C09150=1163.672,78.044,-51.262,-179.316,6.272,148.934
C09151=1163.677,77.794,-51.245,-179.319,6.271,148.934
C09152=1163.682,77.544,-51.228,-179.321,6.270,148.935
C09153=1163.686,77.295,-51.210,-179.324,6.269,148.935
C09154=1163.692,77.046,-51.193,-179.327,6.267,148.936
C09155=1163.696,76.797,-51.177,-179.329,6.266,148.936
C09156=1163.702,76.547,-51.159,-179.332,6.265,148.937
C09157=1163.707,76.298,-51.141,-179.335,6.263,148.937
C09158=1163.711,76.048,-51.125,-179.338,6.263,148.938
C09159=1163.717,75.799,-51.108,-179.340,6.261,148.938
C09160=1163.721,75.550,-51.091,-179.342,6.260,148.939
C09161=1163.727,75.300,-51.074,-179.346,6.259,148.939
C09162=1163.731,75.050,-51.057,-179.348,6.258,148.940
C09163=1163.736,74.801,-51.039,-179.351,6.257,148.940
C09164=1163.741,74.553,-51.023,-179.353,6.256,148.941
C09165=1163.746,74.303,-51.006,-179.356,6.254,148.941
C09166=1163.751,74.053,-50.989,-179.359,6.254,148.942
C09167=1163.755,73.804,-50.972,-179.361,6.252,148.942
C09168=1163.761,73.555,-50.955,-179.364,6.252,148.943
C09169=1163.766,73.305,-50.939,-179.367,6.250,148.944
C09170=1163.771,73.055,-50.922,-179.369,6.249,148.944
C09171=1163.775,72.807,-50.904,-179.372,6.248,148.945
C09172=1163.781,72.557,-50.887,-179.374,6.247,148.945
C09173=1163.785,72.308,-50.871,-179.377,6.246,148.946
C09174=1163.790,72.058,-50.854,-179.380,6.244,148.946
C09175=1163.796,71.809,-50.837,-179.383,6.243,148.947
C09176=1163.800,71.560,-50.820,-179.385,6.242,148.947
C09177=1163.805,71.310,-50.803,-179.388,6.241,148.948
C09178=1163.810,71.061,-50.786,-179.391,6.239,148.948
C09179=1163.815,70.812,-50.770,-179.393,6.239,148.949
C09180=1163.820,70.562,-50.753,-179.396,6.237,148.949
C09181=1163.824,70.313,-50.736,-179.398,6.236,148.950
C09182=1163.830,70.064,-50.720,-179.401,6.235,148.950
C09183=1163.835,69.814,-50.703,-179.404,6.234,148.951
C09184=1163.839,69.564,-50.686,-179.406,6.233,148.951
C09185=1163.844,69.316,-50.670,-179.409,6.232,148.952
C09186=1163.850,69.065,-50.653,-179.412,6.230,148.952
C09187=1163.854,68.816,-50.636,-179.414,6.230,148.953
C09188=1163.859,68.567,-50.620,-179.417,6.228,148.954
C09189=1163.865,68.317,-50.603,-179.419,6.227,148.954
C09190=1163.869,68.068,-50.586,-179.423,6.226,148.955
C09191=1163.874,67.819,-50.570,-179.425,6.225,148.955
C09192=1163.879,67.569,-50.553,-179.427,6.225,148.956
C09193=1163.884,67.320,-50.536,-179.430,6.223,148.956
C09194=1163.889,67.071,-50.520,-179.433,6.222,148.957
C09195=1163.894,66.821,-50.504,-179.435,6.221,148.957
C09196=1163.900,66.572,-50.487,-179.438,6.220,148.958
C09197=1163.904,66.322,-50.470,-179.441,6.219,148.958
C09198=1163.909,66.073,-50.453,-179.443,6.218,148.959
C09199=1163.914,65.824,-50.437,-179.446,6.216,148.959
C09200=1163.919,65.574,-50.420,-179.448,6.215,148.960
C09201=1163.924,65.325,-50.404,-179.452,6.214,148.961
C09202=1163.929,65.075,-50.388,-179.454,6.213,148.961
C09203=1163.933,64.826,-50.371,-179.457,6.212,148.962
C09204=1163.938,64.577,-50.355,-179.459,6.211,148.962
C09205=1163.944,64.327,-50.338,-179.462,6.209,148.962
C09206=1163.949,64.078,-50.322,-179.464,6.209,148.963
C09207=1163.953,63.828,-50.305,-179.467,6.207,148.964
C09208=1163.958,63.579,-50.288,-179.470,6.207,148.964
C09209=1163.963,63.329,-50.273,-179.472,6.206,148.965
C09210=1163.968,63.080,-50.256,-179.475,6.205,148.965
C09211=1163.974,62.831,-50.239,-179.477,6.204,148.966
C09212=1163.978,62.581,-50.223,-179.481,6.202,148.966
C09213=1163.983,62.332,-50.207,-179.483,6.202,148.967
C09214=1163.988,62.082,-50.190,-179.485,6.200,148.967
C09215=1163.993,61.833,-50.175,-179.488,6.199,148.968
C09216=1163.998,61.584,-50.158,-179.491,6.198,148.968
C09217=1164.004,61.334,-50.141,-179.493,6.197,148.969
C09218=1164.008,61.084,-50.125,-179.496,6.195,148.969
C09219=1164.013,60.836,-50.109,-179.499,6.195,148.970
C09220=1164.018,60.585,-50.093,-179.501,6.194,148.971
C09221=1164.023,60.337,-50.077,-179.504,6.193,148.971
C09222=1164.028,60.087,-50.060,-179.506,6.192,148.972
C09223=1164.033,59.837,-50.044,-179.510,6.191,148.972
C09224=1164.038,59.588,-50.028,-179.512,6.190,148.973
C09225=1164.043,59.339,-50.012,-179.514,6.188,148.973
C09226=1164.047,59.089,-49.996,-179.517,6.188,148.974
C09227=1164.053,58.840,-49.980,-179.519,6.187,148.974
C09228=1164.057,58.591,-49.963,-179.522,6.185,148.975
C09229=1164.063,58.341,-49.948,-179.525,6.185,148.975
C09230=1164.068,58.091,-49.930,-179.528,6.183,148.976
C09231=1164.073,57.843,-49.914,-179.530,6.182,148.977
C09232=1164.078,57.592,-49.898,-179.533,6.181,148.977
C09233=1164.083,57.343,-49.883,-179.535,6.180,148.978
C09234=1164.088,57.094,-49.866,-179.538,6.180,148.978
C09235=1164.093,56.844,-49.850,-179.541,6.178,148.979
C09236=1164.098,56.595,-49.834,-179.543,6.178,148.979
C09237=1164.103,56.345,-49.818,-179.546,6.176,148.980
C09238=1164.108,56.097,-49.802,-179.549,6.175,148.981
C09239=1164.113,55.846,-49.786,-179.551,6.174,148.981
C09240=1164.118,55.598,-49.770,-179.554,6.173,148.981
C09241=1164.123,55.348,-49.754,-179.556,6.172,148.982
C09242=1164.128,55.098,-49.738,-179.559,6.171,148.982
C09243=1164.132,54.849,-49.722,-179.562,6.170,148.983
C09244=1164.137,54.600,-49.706,-179.564,6.169,148.984
C09245=1164.143,54.331,-49.689,-179.567,6.168,148.984
C09246=1164.148,54.063,-49.672,-179.570,6.167,148.985
C09247=1164.153,53.793,-49.655,-179.572,6.166,148.985
C09248=1164.159,53.526,-49.637,-179.576,6.165,148.986
C09249=1164.164,53.276,-49.622,-179.578,6.164,148.987
C09250=1164.169,53.026,-49.606,-179.581,6.162,148.987
C09251=1164.174,52.777,-49.589,-179.584,6.162,148.988
C09252=1164.179,52.528,-49.574,-179.586,6.161,148.988
C09253=1164.184,52.278,-49.558,-179.589,6.159,148.989
C09254=1164.189,52.028,-49.542,-179.591,6.159,148.989
C09255=1164.194,51.779,-49.526,-179.593,6.158,148.990
C09256=1164.198,51.530,-49.511,-179.597,6.157,148.990
C09257=1164.204,51.280,-49.495,-179.599,6.156,148.991
C09258=1164.209,51.030,-49.479,-179.602,6.155,148.992
C09259=1164.214,50.782,-49.463,-179.604,6.154,148.992
C09260=1164.219,50.532,-49.447,-179.607,6.153,148.993
C09261=1164.224,50.282,-49.431,-179.610,6.151,148.993
C09262=1164.229,50.033,-49.416,-179.612,6.151,148.994
C09263=1164.234,49.784,-49.400,-179.614,6.150,148.994
C09264=1164.238,49.534,-49.384,-179.618,6.149,148.995
C09265=1164.244,49.285,-49.368,-179.620,6.148,148.995
C09266=1164.249,49.035,-49.353,-179.623,6.147,148.996
C09267=1164.253,48.785,-49.337,-179.625,6.146,148.996
C09268=1164.259,48.536,-49.322,-179.628,6.145,148.997
C09269=1164.264,48.287,-49.305,-179.630,6.144,148.998
C09270=1164.268,48.037,-49.290,-179.633,6.143,148.998
C09271=1164.274,47.788,-49.274,-179.635,6.142,148.999
C09272=1164.279,47.539,-49.259,-179.639,6.141,148.999
C09273=1164.284,47.289,-49.243,-179.641,6.140,149.000
C09274=1164.289,47.039,-49.227,-179.643,6.140,149.000
C09275=1164.294,46.790,-49.212,-179.646,6.138,149.001
C09276=1164.299,46.541,-49.197,-179.649,6.137,149.002
C09277=1164.304,46.291,-49.181,-179.651,6.137,149.002
C09278=1164.309,46.041,-49.165,-179.654,6.135,149.003
C09279=1164.314,45.792,-49.150,-179.656,6.134,149.003
C09280=1164.319,45.543,-49.135,-179.659,6.134,149.004
C09281=1164.323,45.293,-49.118,-179.662,6.132,149.004
C09282=1164.329,45.044,-49.102,-179.664,6.132,149.005
C09283=1164.333,44.795,-49.087,-179.666,6.131,149.005
C09284=1164.339,44.545,-49.072,-179.670,6.130,149.006
C09285=1164.344,44.295,-49.056,-179.672,6.129,149.006
C09286=1164.348,44.046,-49.041,-179.674,6.128,149.007
C09287=1164.354,43.796,-49.026,-179.677,6.127,149.008
C09288=1164.359,43.547,-49.010,-179.680,6.126,149.008
C09289=1164.364,43.298,-48.995,-179.682,6.125,149.009
C09290=1164.369,43.047,-48.980,-179.685,6.124,149.009
C09291=1164.374,42.798,-48.964,-179.687,6.123,149.010
C09292=1164.379,42.549,-48.949,-179.690,6.123,149.011
C09293=1164.384,42.300,-48.933,-179.693,6.121,149.011
C09294=1164.389,42.050,-48.918,-179.695,6.121,149.012
C09295=1164.394,41.800,-48.902,-179.698,6.120,149.012
C09296=1164.399,41.551,-48.887,-179.701,6.118,149.013
C09297=1164.404,41.302,-48.872,-179.703,6.118,149.013
C09298=1164.409,41.052,-48.856,-179.706,6.117,149.014
C09299=1164.414,40.803,-48.842,-179.708,6.115,149.014
C09300=1164.419,40.553,-48.826,-179.711,6.115,149.015
C09301=1164.424,40.303,-48.810,-179.713,6.114,149.015
C09302=1164.429,40.054,-48.795,-179.716,6.113,149.016
C09303=1164.434,39.805,-48.780,-179.719,6.112,149.017
C09304=1164.439,39.556,-48.765,-179.721,6.111,149.017
C09305=1164.445,39.306,-48.750,-179.724,6.111,149.018
C09306=1164.449,39.057,-48.735,-179.727,6.109,149.018
C09307=1164.454,38.806,-48.719,-179.729,6.109,149.019
C09308=1164.459,38.557,-48.704,-179.731,6.108,149.019
C09309=1164.464,38.308,-48.688,-179.735,6.107,149.020
C09310=1164.470,38.058,-48.674,-179.737,6.106,149.021
C09311=1164.474,37.809,-48.659,-179.739,6.105,149.021
C09312=1164.480,37.559,-48.643,-179.742,6.104,149.022
C09313=1164.484,37.310,-48.628,-179.745,6.103,149.022
C09314=1164.490,37.060,-48.613,-179.747,6.102,149.023
C09315=1164.494,36.811,-48.598,-179.750,6.102,149.023
C09316=1164.500,36.561,-48.582,-179.752,6.100,149.024
C09317=1164.505,36.311,-48.568,-179.755,6.100,149.025
C09318=1164.509,36.062,-48.553,-179.757,6.099,149.025
C09319=1164.515,35.813,-48.537,-179.760,6.098,149.026
C09320=1164.519,35.564,-48.522,-179.763,6.097,149.026
C09321=1164.525,35.314,-48.507,-179.765,6.096,149.027
C09322=1164.530,35.065,-48.492,-179.767,6.095,149.027
C09323=1164.535,34.815,-48.478,-179.771,6.094,149.028
C09324=1164.540,34.566,-48.463,-179.773,6.094,149.029
C09325=1164.545,34.316,-48.447,-179.775,6.093,149.029
C09326=1164.550,34.066,-48.433,-179.778,6.092,149.030
C09327=1164.555,33.817,-48.418,-179.781,6.091,149.030
C09328=1164.560,33.567,-48.402,-179.783,6.090,149.031
C09329=1164.565,33.318,-48.387,-179.786,6.089,149.031
C09330=1164.570,33.068,-48.372,-179.789,6.088,149.032
C09331=1164.575,32.818,-48.358,-179.791,6.087,149.032
C09332=1164.580,32.569,-48.343,-179.794,6.087,149.033
C09333=1164.585,32.319,-48.328,-179.796,6.086,149.034
C09334=1164.590,32.070,-48.313,-179.799,6.085,149.034
C09335=1164.595,31.821,-48.298,-179.801,6.084,149.035
C09336=1164.600,31.571,-48.283,-179.804,6.083,149.035
C09337=1164.605,31.322,-48.268,-179.806,6.082,149.036
C09338=1164.611,31.072,-48.253,-179.809,6.081,149.037
C09339=1164.615,30.823,-48.238,-179.812,6.081,149.037
C09340=1164.620,30.573,-48.224,-179.814,6.080,149.038
C09341=1164.625,30.324,-48.209,-179.817,6.079,149.038
C09342=1164.631,30.074,-48.194,-179.819,6.078,149.039
C09343=1164.635,29.825,-48.179,-179.822,6.077,149.039
C09344=1164.640,29.575,-48.165,-179.824,6.076,149.040
C09345=1164.646,29.325,-48.150,-179.827,6.076,149.041
C09346=1164.651,29.076,-48.135,-179.830,6.074,149.041
C09347=1164.655,28.827,-48.120,-179.832,6.074,149.042
C09348=1164.661,28.577,-48.105,-179.834,6.073,149.042
C09349=1164.666,28.308,-48.089,-179.837,6.072,149.043
C09350=1164.671,28.040,-48.073,-179.840,6.071,149.044
C09351=1164.677,27.770,-48.057,-179.843,6.071,149.044
C09352=1164.683,27.502,-48.042,-179.846,6.069,149.045
C09353=1164.688,27.253,-48.028,-179.848,6.068,149.045
C09354=1164.693,27.003,-48.013,-179.851,6.068,149.046
C09355=1164.698,26.754,-47.998,-179.853,6.067,149.046
C09356=1164.703,26.504,-47.983,-179.856,6.066,149.047
C09357=1164.708,26.254,-47.969,-179.859,6.065,149.048
C09358=1164.713,26.005,-47.954,-179.861,6.065,149.048
C09359=1164.718,25.755,-47.939,-179.863,6.064,149.049
C09360=1164.723,25.505,-47.925,-179.866,6.063,149.049
C09361=1164.728,25.256,-47.910,-179.869,6.062,149.050
C09362=1164.733,25.006,-47.896,-179.871,6.061,149.051
C09363=1164.738,24.757,-47.881,-179.874,6.060,149.051
C09364=1164.743,24.507,-47.867,-179.876,6.060,149.052
C09365=1164.749,24.258,-47.852,-179.879,6.059,149.052
C09366=1164.754,24.009,-47.838,-179.882,6.058,149.053
C09367=1164.759,23.759,-47.823,-179.884,6.057,149.054
C09368=1164.763,23.510,-47.808,-179.887,6.056,149.054
C09369=1164.768,23.260,-47.794,-179.889,6.056,149.055
C09370=1164.773,23.010,-47.780,-179.891,6.055,149.055
C09371=1164.779,22.760,-47.765,-179.895,6.054,149.056
C09372=1164.784,22.511,-47.751,-179.897,6.053,149.056
C09373=1164.788,22.262,-47.736,-179.899,6.052,149.057
C09374=1164.794,22.013,-47.722,-179.902,6.052,149.057
C09375=1164.799,21.763,-47.708,-179.904,6.051,149.058
C09376=1164.804,21.513,-47.693,-179.907,6.050,149.059
C09377=1164.809,21.263,-47.679,-179.910,6.049,149.059
C09378=1164.814,21.014,-47.665,-179.912,6.049,149.060
C09379=1164.818,20.765,-47.650,-179.914,6.048,149.060
C09380=1164.824,20.516,-47.636,-179.917,6.047,149.061
C09381=1164.830,20.266,-47.621,-179.920,6.046,149.061
C09382=1164.835,20.016,-47.607,-179.922,6.045,149.062
C09383=1164.840,19.766,-47.592,-179.925,6.045,149.063
C09384=1164.845,19.516,-47.578,-179.927,6.044,149.063
C09385=1164.850,19.267,-47.564,-179.930,6.043,149.064
C09386=1164.855,19.018,-47.550,-179.933,6.042,149.064
C09387=1164.860,18.768,-47.536,-179.935,6.041,149.065
C09388=1164.865,18.519,-47.521,-179.937,6.040,149.066
C09389=1164.870,18.269,-47.506,-179.940,6.040,149.066
C09390=1164.875,18.020,-47.492,-179.942,6.039,149.067
C09391=1164.880,17.771,-47.478,-179.945,6.039,149.067
C09392=1164.885,17.521,-47.464,-179.948,6.037,149.068
C09393=1164.890,17.271,-47.450,-179.950,6.037,149.068
C09394=1164.895,17.021,-47.435,-179.953,6.036,149.069
C09395=1164.900,16.772,-47.421,-179.955,6.035,149.070
C09396=1164.906,16.523,-47.407,-179.958,6.035,149.070
C09397=1164.911,16.273,-47.393,-179.960,6.034,149.071
C09398=1164.915,16.023,-47.379,-179.963,6.033,149.071
C09399=1164.920,15.774,-47.364,-179.965,6.032,149.072
C09400=1164.926,15.525,-47.350,-179.968,6.031,149.073
C09401=1164.931,15.275,-47.336,-179.971,6.031,149.073
C09402=1164.936,15.025,-47.322,-179.973,6.030,149.074
C09403=1164.941,14.775,-47.308,-179.976,6.030,149.074
C09404=1164.947,14.526,-47.294,-179.978,6.029,149.075
C09405=1164.951,14.276,-47.281,-179.981,6.027,149.076
C09406=1164.956,14.027,-47.266,-179.983,6.027,149.076
C09407=1164.961,13.777,-47.252,-179.986,6.026,149.077
C09408=1164.966,13.528,-47.238,-179.988,6.026,149.077
C09409=1164.971,13.278,-47.224,-179.991,6.025,149.078
C09410=1164.976,13.029,-47.210,-179.993,6.024,149.079
C09411=1164.982,12.780,-47.196,-179.995,6.024,149.079
C09412=1164.987,12.530,-47.181,-179.999,6.022,149.080
C09413=1164.992,12.279,-47.168,179.999,6.021,149.080
C09414=1164.996,12.030,-47.154,179.997,6.021,149.081
C09415=1165.002,11.781,-47.140,179.994,6.021,149.081
C09416=1165.007,11.531,-47.126,179.992,6.020,149.082
C09417=1165.012,11.282,-47.112,179.989,6.019,149.083
C09418=1165.017,11.033,-47.098,179.987,6.018,149.083
C09419=1165.023,10.782,-47.084,179.984,6.017,149.084
C09420=1165.028,10.533,-47.070,179.981,6.016,149.084
C09421=1165.032,10.284,-47.057,179.979,6.016,149.085
C09422=1165.037,10.034,-47.042,179.976,6.015,149.086
C09423=1165.043,9.784,-47.029,179.974,6.015,149.086
C09424=1165.048,9.535,-47.015,179.971,6.014,149.087
C09425=1165.053,9.285,-47.001,179.969,6.013,149.087
C09426=1165.057,9.036,-46.987,179.967,6.013,149.088
C09427=1165.063,8.786,-46.974,179.964,6.011,149.088
C09428=1165.068,8.536,-46.960,179.961,6.011,149.089
C09429=1165.073,8.287,-46.945,179.958,6.010,149.090
C09430=1165.079,8.038,-46.931,179.956,6.009,149.090
C09431=1165.083,7.788,-46.918,179.954,6.009,149.091
C09432=1165.089,7.539,-46.904,179.951,6.008,149.091
C09433=1165.094,7.289,-46.890,179.949,6.008,149.092
C09434=1165.099,7.039,-46.877,179.947,6.007,149.092
C09435=1165.104,6.790,-46.863,179.944,6.006,149.093
C09436=1165.109,6.540,-46.849,179.941,6.005,149.094
C09437=1165.114,6.290,-46.835,179.939,6.004,149.094
C09438=1165.120,6.041,-46.822,179.936,6.004,149.095
C09439=1165.124,5.791,-46.808,179.934,6.003,149.095
C09440=1165.130,5.542,-46.795,179.931,6.003,149.096
C09441=1165.135,5.292,-46.780,179.929,6.002,149.097
C09442=1165.139,5.042,-46.767,179.926,6.001,149.097
C09443=1165.145,4.793,-46.754,179.924,6.001,149.098
C09444=1165.150,4.543,-46.739,179.921,6.000,149.098
C09445=1165.155,4.294,-46.727,179.919,5.999,149.099
C09446=1165.160,4.044,-46.712,179.917,5.999,149.100
C09447=1165.166,3.795,-46.699,179.913,5.997,149.100
C09448=1165.170,3.545,-46.685,179.911,5.997,149.101
C09449=1165.175,3.295,-46.672,179.909,5.996,149.101
C09450=1165.181,3.046,-46.658,179.906,5.996,149.102
C09451=1165.185,2.797,-46.644,179.904,5.995,149.103
C09452=1165.191,2.547,-46.631,179.901,5.994,149.103
C09453=1165.196,2.278,-46.616,179.898,5.994,149.104
C09454=1165.201,2.008,-46.601,179.896,5.993,149.104
C09455=1165.207,1.739,-46.588,179.893,5.992,149.105
C09456=1165.213,1.470,-46.573,179.890,5.991,149.106
C09457=1165.217,1.220,-46.559,179.888,5.991,149.106
C09458=1165.223,0.971,-46.546,179.886,5.990,149.107
C09459=1165.228,0.720,-46.532,179.883,5.990,149.108
C09460=1165.233,0.471,-46.519,179.881,5.989,149.108
C09461=1165.238,0.221,-46.506,179.878,5.988,149.109
C09462=1165.243,-0.028,-46.492,179.876,5.988,149.109
C09463=1165.248,-0.278,-46.479,179.873,5.987,149.110
C09464=1165.254,-0.527,-46.465,179.871,5.987,149.111
C09465=1165.259,-0.777,-46.451,179.868,5.985,149.111
C09466=1165.264,-1.026,-46.439,179.865,5.985,149.112
C09467=1165.269,-1.276,-46.424,179.863,5.984,149.112
C09468=1165.274,-1.525,-46.412,179.860,5.983,149.113
C09469=1165.279,-1.775,-46.397,179.858,5.983,149.114
C09470=1165.284,-2.024,-46.385,179.856,5.982,149.114
C09471=1165.289,-2.275,-46.371,179.853,5.982,149.115
C09472=1165.294,-2.523,-46.358,179.851,5.981,149.115
C09473=1165.299,-2.774,-46.344,179.848,5.980,149.116
C09474=1165.305,-3.023,-46.332,179.846,5.979,149.116
C09475=1165.310,-3.272,-46.318,179.843,5.979,149.117
C09476=1165.315,-3.522,-46.305,179.841,5.979,149.118
C09477=1165.321,-3.772,-46.292,179.838,5.978,149.118
C09478=1165.325,-4.021,-46.278,179.836,5.977,149.119
C09479=1165.331,-4.271,-46.265,179.834,5.976,149.119
C09480=1165.335,-4.521,-46.252,179.831,5.976,149.120
C09481=1165.341,-4.770,-46.239,179.829,5.975,149.121
C09482=1165.345,-5.020,-46.225,179.826,5.975,149.121
C09483=1165.351,-5.269,-46.212,179.823,5.974,149.122
C09484=1165.356,-5.519,-46.199,179.821,5.973,149.122
C09485=1165.361,-5.769,-46.186,179.819,5.973,149.123
C09486=1165.366,-6.018,-46.172,179.816,5.971,149.124
C09487=1165.372,-6.268,-46.159,179.813,5.971,149.124
C09488=1165.377,-6.517,-46.146,179.810,5.970,149.125
C09489=1165.382,-6.767,-46.134,179.808,5.970,149.125
C09490=1165.387,-7.016,-46.119,179.806,5.969,149.126
C09491=1165.392,-7.266,-46.107,179.803,5.968,149.127
C09492=1165.397,-7.516,-46.093,179.801,5.968,149.127
C09493=1165.402,-7.765,-46.081,179.799,5.967,149.128
C09494=1165.407,-8.015,-46.068,179.796,5.967,149.128
C09495=1165.413,-8.265,-46.054,179.793,5.966,149.129
C09496=1165.417,-8.514,-46.041,179.791,5.965,149.130
C09497=1165.422,-8.764,-46.028,179.789,5.965,149.130
C09498=1165.428,-9.013,-46.015,179.786,5.964,149.131
C09499=1165.433,-9.263,-46.002,179.784,5.964,149.131
C09500=1165.438,-9.513,-45.989,179.781,5.963,149.132
C09501=1165.443,-9.762,-45.976,179.779,5.962,149.133
C09502=1165.448,-10.012,-45.964,179.776,5.962,149.133
C09503=1165.454,-10.262,-45.950,179.774,5.961,149.134
C09504=1165.459,-10.511,-45.937,179.771,5.961,149.134
C09505=1165.464,-10.760,-45.924,179.769,5.960,149.135
C09506=1165.469,-11.010,-45.910,179.767,5.959,149.136
C09507=1165.474,-11.260,-45.898,179.764,5.959,149.136
C09508=1165.479,-11.509,-45.885,179.762,5.958,149.137
C09509=1165.484,-11.759,-45.872,179.759,5.958,149.137
C09510=1165.490,-12.009,-45.859,179.757,5.957,149.138
C09511=1165.495,-12.258,-45.847,179.754,5.956,149.139
C09512=1165.499,-12.508,-45.834,179.752,5.956,149.139
C09513=1165.505,-12.758,-45.820,179.749,5.955,149.140
C09514=1165.510,-13.007,-45.808,179.747,5.955,149.140
C09515=1165.515,-13.257,-45.795,179.745,5.954,149.141
C09516=1165.520,-13.506,-45.782,179.742,5.953,149.142
C09517=1165.526,-13.756,-45.769,179.739,5.953,149.142
C09518=1165.530,-14.006,-45.756,179.737,5.952,149.143
C09519=1165.535,-14.255,-45.743,179.734,5.952,149.143
C09520=1165.540,-14.505,-45.731,179.732,5.951,149.144
C09521=1165.546,-14.754,-45.718,179.730,5.950,149.145
C09522=1165.551,-15.004,-45.705,179.727,5.950,149.145
C09523=1165.556,-15.254,-45.692,179.725,5.949,149.146
C09524=1165.561,-15.503,-45.679,179.722,5.949,149.146
C09525=1165.567,-15.753,-45.667,179.720,5.948,149.147
C09526=1165.572,-16.003,-45.654,179.717,5.948,149.148
C09527=1165.577,-16.252,-45.641,179.715,5.947,149.148
C09528=1165.582,-16.502,-45.629,179.712,5.946,149.149
C09529=1165.587,-16.751,-45.616,179.710,5.946,149.149
C09530=1165.592,-17.001,-45.603,179.708,5.945,149.150
C09531=1165.598,-17.251,-45.590,179.705,5.945,149.151
C09532=1165.603,-17.500,-45.577,179.703,5.944,149.151
C09533=1165.608,-17.750,-45.566,179.701,5.944,149.152
C09534=1165.613,-18.000,-45.553,179.698,5.943,149.152
C09535=1165.618,-18.249,-45.540,179.696,5.943,149.153
C09536=1165.624,-18.499,-45.527,179.693,5.942,149.154
C09537=1165.629,-18.748,-45.514,179.691,5.942,149.154
C09538=1165.634,-18.998,-45.502,179.688,5.941,149.155
C09539=1165.639,-19.248,-45.489,179.686,5.940,149.155
C09540=1165.644,-19.498,-45.477,179.683,5.940,149.156
C09541=1165.649,-19.747,-45.464,179.681,5.939,149.157
C09542=1165.654,-19.996,-45.452,179.679,5.939,149.157
C09543=1165.660,-20.246,-45.438,179.676,5.938,149.158
C09544=1165.665,-20.496,-45.426,179.674,5.937,149.158
C09545=1165.670,-20.746,-45.413,179.671,5.937,149.159
C09546=1165.675,-20.995,-45.401,179.669,5.936,149.159
C09547=1165.680,-21.244,-45.388,179.666,5.936,149.160
C09548=1165.686,-21.494,-45.376,179.664,5.935,149.161
C09549=1165.690,-21.744,-45.363,179.661,5.934,149.161
C09550=1165.695,-21.994,-45.351,179.659,5.934,149.162
C09551=1165.701,-22.244,-45.339,179.657,5.933,149.162
C09552=1165.706,-22.493,-45.326,179.654,5.933,149.163
C09553=1165.711,-22.742,-45.314,179.651,5.932,149.164
C09554=1165.716,-22.992,-45.302,179.649,5.931,149.164
C09555=1165.722,-23.242,-45.289,179.647,5.932,149.165
C09556=1165.727,-23.492,-45.276,179.645,5.931,149.166
C09557=1165.733,-23.761,-45.263,179.642,5.931,149.166
C09558=1165.738,-24.031,-45.249,179.639,5.929,149.167
C09559=1165.744,-24.302,-45.236,179.636,5.929,149.168
C09560=1165.749,-24.571,-45.223,179.634,5.928,149.168
C09561=1165.754,-24.820,-45.210,179.631,5.928,149.169
C09562=1165.760,-25.070,-45.198,179.629,5.927,149.169
C09563=1165.764,-25.320,-45.185,179.627,5.926,149.170
C09564=1165.770,-25.570,-45.173,179.625,5.927,149.171
C09565=1165.775,-25.819,-45.161,179.622,5.926,149.171
C09566=1165.780,-26.069,-45.148,179.620,5.926,149.172
C09567=1165.785,-26.319,-45.136,179.617,5.925,149.173
C09568=1165.791,-26.568,-45.124,179.615,5.924,149.173
C09569=1165.796,-26.818,-45.112,179.612,5.924,149.174
C09570=1165.801,-27.067,-45.099,179.610,5.923,149.174
C09571=1165.807,-27.317,-45.087,179.607,5.923,149.175
C09572=1165.811,-27.566,-45.075,179.605,5.922,149.175
C09573=1165.815,-27.816,-45.062,179.602,5.921,149.176
C09574=1165.821,-28.066,-45.050,179.600,5.921,149.177
C09575=1165.826,-28.315,-45.038,179.598,5.920,149.177
C09576=1165.831,-28.565,-45.026,179.596,5.921,149.178
C09577=1165.837,-28.815,-45.013,179.593,5.920,149.178
C09578=1165.842,-29.065,-45.001,179.591,5.919,149.179
C09579=1165.847,-29.314,-44.989,179.589,5.918,149.180
C09580=1165.853,-29.564,-44.977,179.586,5.918,149.180
C09581=1165.858,-29.814,-44.965,179.583,5.918,149.181
C09582=1165.863,-30.063,-44.952,179.581,5.917,149.181
C09583=1165.868,-30.313,-44.941,179.578,5.916,149.182
C09584=1165.873,-30.562,-44.928,179.576,5.916,149.183
C09585=1165.878,-30.812,-44.917,179.574,5.915,149.183
C09586=1165.883,-31.061,-44.904,179.571,5.915,149.184
C09587=1165.889,-31.311,-44.892,179.569,5.915,149.184
C09588=1165.894,-31.561,-44.879,179.567,5.914,149.185
C09589=1165.899,-31.811,-44.868,179.564,5.913,149.186
C09590=1165.904,-32.060,-44.856,179.562,5.913,149.186
C09591=1165.909,-32.309,-44.844,179.560,5.912,149.187
C09592=1165.915,-32.559,-44.832,179.557,5.912,149.187
C09593=1165.920,-32.809,-44.820,179.554,5.911,149.188
C09594=1165.925,-33.059,-44.807,179.552,5.911,149.189
C09595=1165.931,-33.309,-44.795,179.549,5.910,149.189
C09596=1165.935,-33.558,-44.783,179.548,5.910,149.190
C09597=1165.940,-33.808,-44.772,179.545,5.910,149.190
C09598=1165.946,-34.058,-44.760,179.543,5.909,149.191
C09599=1165.951,-34.307,-44.747,179.540,5.908,149.192
C09600=1165.956,-34.557,-44.735,179.538,5.908,149.192
C09601=1165.961,-34.806,-44.724,179.536,5.907,149.193
C09602=1165.967,-35.056,-44.712,179.533,5.907,149.194
C09603=1165.972,-35.306,-44.699,179.531,5.906,149.194
C09604=1165.977,-35.556,-44.688,179.529,5.906,149.195
C09605=1165.983,-35.806,-44.676,179.526,5.906,149.195
C09606=1165.987,-36.055,-44.664,179.524,5.905,149.196
C09607=1165.992,-36.304,-44.652,179.521,5.905,149.197
C09608=1165.998,-36.554,-44.640,179.519,5.904,149.197
C09609=1166.003,-36.804,-44.628,179.516,5.903,149.198
C09610=1166.008,-37.053,-44.616,179.514,5.903,149.198
C09611=1166.013,-37.303,-44.604,179.511,5.902,149.199
C09612=1166.018,-37.553,-44.592,179.510,5.902,149.199
C09613=1166.023,-37.803,-44.581,179.507,5.902,149.200
C09614=1166.028,-38.052,-44.568,179.504,5.901,149.201
C09615=1166.034,-38.301,-44.557,179.502,5.901,149.201
C09616=1166.040,-38.551,-44.545,179.500,5.900,149.202
C09617=1166.044,-38.801,-44.534,179.497,5.899,149.202
C09618=1166.050,-39.051,-44.522,179.495,5.899,149.203
C09619=1166.055,-39.301,-44.510,179.493,5.899,149.204
C09620=1166.060,-39.550,-44.498,179.491,5.898,149.204
C09621=1166.065,-39.800,-44.486,179.488,5.898,149.205
C09622=1166.071,-40.050,-44.474,179.486,5.897,149.206
C09623=1166.075,-40.299,-44.463,179.483,5.897,149.206
C09624=1166.081,-40.549,-44.451,179.481,5.896,149.207
C09625=1166.087,-40.799,-44.439,179.479,5.896,149.207
C09626=1166.091,-41.048,-44.428,179.477,5.896,149.208
C09627=1166.097,-41.297,-44.415,179.474,5.895,149.209
C09628=1166.102,-41.547,-44.404,179.471,5.895,149.209
C09629=1166.107,-41.797,-44.392,179.469,5.894,149.210
C09630=1166.112,-42.047,-44.380,179.466,5.894,149.210
C09631=1166.117,-42.297,-44.369,179.464,5.893,149.211
C09632=1166.122,-42.547,-44.357,179.462,5.893,149.212
C09633=1166.128,-42.796,-44.346,179.460,5.892,149.212
C09634=1166.133,-43.045,-44.334,179.457,5.892,149.213
C09635=1166.138,-43.295,-44.323,179.455,5.891,149.213
C09636=1166.144,-43.545,-44.311,179.452,5.891,149.214
C09637=1166.148,-43.795,-44.299,179.450,5.890,149.215
C09638=1166.154,-44.045,-44.287,179.448,5.890,149.215
C09639=1166.159,-44.294,-44.277,179.446,5.890,149.216
C09640=1166.165,-44.544,-44.265,179.443,5.889,149.216
C09641=1166.169,-44.793,-44.253,179.441,5.889,149.217
C09642=1166.175,-45.043,-44.242,179.438,5.888,149.217
C09643=1166.180,-45.293,-44.230,179.436,5.887,149.218
C09644=1166.185,-45.543,-44.218,179.434,5.888,149.219
C09645=1166.191,-45.792,-44.207,179.432,5.887,149.219
C09646=1166.196,-46.042,-44.196,179.429,5.887,149.220
C09647=1166.201,-46.292,-44.184,179.427,5.886,149.221
C09648=1166.206,-46.541,-44.172,179.424,5.885,149.221
C09649=1166.211,-46.791,-44.160,179.422,5.885,149.222
C09650=1166.216,-47.040,-44.150,179.420,5.885,149.222
C09651=1166.222,-47.290,-44.138,179.418,5.884,149.223
C09652=1166.227,-47.540,-44.126,179.415,5.884,149.224
C09653=1166.232,-47.790,-44.114,179.412,5.883,149.224
C09654=1166.237,-48.039,-44.103,179.410,5.882,149.225
C09655=1166.243,-48.288,-44.092,179.408,5.883,149.225
C09656=1166.248,-48.539,-44.081,179.406,5.882,149.226
C09657=1166.253,-48.789,-44.069,179.403,5.882,149.227
C09658=1166.258,-49.038,-44.058,179.401,5.881,149.227
C09659=1166.264,-49.287,-44.046,179.398,5.880,149.228
C09660=1166.269,-49.537,-44.035,179.397,5.880,149.228
C09661=1166.274,-49.808,-44.023,179.394,5.880,149.229
C09662=1166.280,-50.078,-44.010,179.391,5.880,149.230
C09663=1166.286,-50.349,-43.998,179.389,5.879,149.230
C09664=1166.291,-50.620,-43.986,179.386,5.879,149.231
C09665=1166.297,-50.869,-43.975,179.384,5.878,149.232
C09666=1166.302,-51.119,-43.963,179.381,5.878,149.232
C09667=1166.307,-51.368,-43.952,179.379,5.877,149.233
C09668=1166.312,-51.618,-43.940,179.377,5.877,149.233
C09669=1166.318,-51.868,-43.930,179.375,5.876,149.234
C09670=1166.322,-52.117,-43.918,179.372,5.876,149.235
C09671=1166.328,-52.367,-43.906,179.370,5.875,149.235
C09672=1166.333,-52.616,-43.895,179.367,5.875,149.236
C09673=1166.339,-52.867,-43.884,179.366,5.875,149.236
C09674=1166.344,-53.116,-43.873,179.363,5.874,149.237
C09675=1166.348,-53.366,-43.862,179.360,5.874,149.238
C09676=1166.354,-53.615,-43.850,179.358,5.873,149.238
C09677=1166.359,-53.865,-43.840,179.356,5.873,149.239
C09678=1166.364,-54.115,-43.828,179.354,5.873,149.239
C09679=1166.370,-54.364,-43.817,179.351,5.872,149.240
C09680=1166.375,-54.614,-43.806,179.349,5.871,149.241
C09681=1166.380,-54.864,-43.795,179.346,5.871,149.241
C09682=1166.386,-55.113,-43.783,179.345,5.871,149.242
C09683=1166.390,-55.363,-43.772,179.342,5.871,149.242
C09684=1166.395,-55.613,-43.762,179.340,5.870,149.243
C09685=1166.401,-55.862,-43.750,179.337,5.869,149.244
C09686=1166.406,-56.112,-43.739,179.335,5.870,149.244
C09687=1166.411,-56.362,-43.728,179.333,5.869,149.245
C09688=1166.417,-56.612,-43.717,179.330,5.869,149.246
C09689=1166.422,-56.861,-43.705,179.328,5.868,149.246
C09690=1166.427,-57.111,-43.695,179.325,5.867,149.247
C09691=1166.433,-57.361,-43.683,179.324,5.867,149.247
C09692=1166.438,-57.610,-43.672,179.321,5.867,149.248
C09693=1166.443,-57.861,-43.661,179.319,5.866,149.248
C09694=1166.448,-58.110,-43.650,179.316,5.866,149.249
C09695=1166.454,-58.360,-43.639,179.315,5.866,149.250
C09696=1166.458,-58.610,-43.628,179.312,5.865,149.250
C09697=1166.464,-58.859,-43.617,179.310,5.865,149.251
C09698=1166.469,-59.109,-43.607,179.307,5.864,149.251
C09699=1166.474,-59.359,-43.595,179.305,5.865,149.252
C09700=1166.480,-59.608,-43.584,179.303,5.864,149.253
C09701=1166.484,-59.858,-43.573,179.300,5.863,149.253
C09702=1166.490,-60.108,-43.563,179.298,5.863,149.254
C09703=1166.495,-60.357,-43.551,179.296,5.863,149.255
C09704=1166.500,-60.607,-43.540,179.294,5.862,149.255
C09705=1166.506,-60.857,-43.530,179.291,5.862,149.256
C09706=1166.510,-61.106,-43.518,179.289,5.861,149.256
C09707=1166.516,-61.356,-43.508,179.287,5.861,149.257
C09708=1166.521,-61.606,-43.496,179.285,5.861,149.257
C09709=1166.526,-61.856,-43.486,179.282,5.860,149.258
C09710=1166.532,-62.105,-43.475,179.280,5.859,149.259
C09711=1166.537,-62.355,-43.464,179.278,5.860,149.259
C09712=1166.542,-62.604,-43.453,179.276,5.859,149.260
C09713=1166.548,-62.855,-43.442,179.273,5.859,149.260
C09714=1166.553,-63.104,-43.432,179.271,5.858,149.261
C09715=1166.558,-63.354,-43.421,179.269,5.858,149.262
C09716=1166.563,-63.604,-43.410,179.266,5.858,149.262
C09717=1166.568,-63.853,-43.399,179.264,5.857,149.263
C09718=1166.573,-64.103,-43.388,179.261,5.857,149.264
C09719=1166.579,-64.352,-43.377,179.260,5.857,149.264
C09720=1166.584,-64.603,-43.366,179.257,5.856,149.265
C09721=1166.590,-64.852,-43.355,179.255,5.855,149.265
C09722=1166.595,-65.102,-43.345,179.252,5.855,149.266
C09723=1166.600,-65.351,-43.335,179.250,5.855,149.266
C09724=1166.605,-65.601,-43.323,179.248,5.855,149.267
C09725=1166.610,-65.851,-43.313,179.246,5.854,149.268
C09726=1166.615,-66.101,-43.303,179.244,5.854,149.268
C09727=1166.621,-66.350,-43.291,179.241,5.853,149.269
C09728=1166.626,-66.600,-43.280,179.239,5.853,149.269
C09729=1166.631,-66.850,-43.269,179.236,5.852,149.270
C09730=1166.637,-67.099,-43.259,179.234,5.853,149.271
C09731=1166.642,-67.350,-43.248,179.232,5.852,149.271
C09732=1166.647,-67.599,-43.237,179.230,5.851,149.272
C09733=1166.652,-67.849,-43.227,179.227,5.851,149.272
C09734=1166.658,-68.098,-43.217,179.225,5.851,149.273
C09735=1166.662,-68.348,-43.205,179.223,5.850,149.273
C09736=1166.668,-68.598,-43.195,179.220,5.850,149.274
C09737=1166.674,-68.847,-43.185,179.219,5.850,149.275
C09738=1166.679,-69.097,-43.174,179.216,5.849,149.275
C09739=1166.685,-69.347,-43.163,179.214,5.849,149.276
C09740=1166.690,-69.597,-43.152,179.211,5.848,149.277
C09741=1166.695,-69.846,-43.142,179.210,5.848,149.277
C09742=1166.700,-70.097,-43.132,179.207,5.848,149.278
C09743=1166.705,-70.346,-43.121,179.205,5.847,149.278
C09744=1166.710,-70.596,-43.110,179.203,5.847,149.279
C09745=1166.716,-70.845,-43.100,179.201,5.847,149.279
C09746=1166.721,-71.096,-43.089,179.198,5.846,149.280
C09747=1166.726,-71.345,-43.078,179.196,5.846,149.281
C09748=1166.731,-71.595,-43.068,179.194,5.846,149.281
C09749=1166.737,-71.844,-43.058,179.191,5.845,149.282
C09750=1166.743,-72.094,-43.047,179.189,5.845,149.282
C09751=1166.747,-72.343,-43.036,179.187,5.845,149.283
C09752=1166.753,-72.593,-43.026,179.185,5.844,149.284
C09753=1166.758,-72.843,-43.015,179.182,5.844,149.284
C09754=1166.763,-73.093,-43.005,179.180,5.844,149.285
C09755=1166.768,-73.343,-42.994,179.178,5.843,149.285
C09756=1166.774,-73.593,-42.984,179.175,5.843,149.286
C09757=1166.779,-73.842,-42.973,179.174,5.843,149.287
C09758=1166.784,-74.092,-42.963,179.171,5.842,149.287
C09759=1166.790,-74.341,-42.953,179.169,5.842,149.288
C09760=1166.794,-74.591,-42.943,179.167,5.842,149.288
C09761=1166.800,-74.841,-42.932,179.165,5.841,149.289
C09762=1166.805,-75.090,-42.922,179.162,5.841,149.290
C09763=1166.810,-75.341,-42.912,179.160,5.840,149.290
C09764=1166.816,-75.590,-42.901,179.158,5.840,149.291
C09765=1166.822,-75.861,-42.889,179.155,5.840,149.292
C09766=1166.827,-76.132,-42.879,179.153,5.839,149.292
C09767=1166.833,-76.403,-42.867,179.150,5.839,149.293
C09768=1166.838,-76.675,-42.856,179.148,5.838,149.293
C09769=1166.844,-76.924,-42.846,179.146,5.838,149.294
C09770=1166.849,-77.174,-42.835,179.143,5.838,149.295
C09771=1166.855,-77.424,-42.825,179.141,5.837,149.295
C09772=1166.860,-77.673,-42.815,179.139,5.838,149.296
C09773=1166.865,-77.924,-42.804,179.137,5.837,149.296
C09774=1166.871,-78.173,-42.794,179.134,5.836,149.297
C09775=1166.876,-78.423,-42.784,179.133,5.836,149.297
C09776=1166.881,-78.673,-42.773,179.130,5.836,149.298
C09777=1166.886,-78.922,-42.764,179.128,5.835,149.299
C09778=1166.892,-79.172,-42.753,179.126,5.836,149.299
C09779=1166.897,-79.422,-42.743,179.123,5.835,149.300
C09780=1166.903,-79.672,-42.733,179.121,5.835,149.301
C09781=1166.908,-79.921,-42.722,179.119,5.835,149.301
C09782=1166.913,-80.171,-42.712,179.116,5.834,149.302
C09783=1166.918,-80.421,-42.702,179.114,5.833,149.302
C09784=1166.924,-80.670,-42.692,179.113,5.833,149.303
C09785=1166.929,-80.920,-42.682,179.110,5.833,149.303
C09786=1166.934,-81.170,-42.671,179.108,5.832,149.304
C09787=1166.940,-81.419,-42.661,179.106,5.833,149.305
C09788=1166.944,-81.669,-42.651,179.104,5.832,149.305
C09789=1166.950,-81.919,-42.641,179.101,5.831,149.306
C09790=1166.955,-82.169,-42.631,179.099,5.831,149.306
C09791=1166.961,-82.418,-42.621,179.097,5.831,149.307
C09792=1166.966,-82.668,-42.610,179.094,5.830,149.307
C09793=1166.971,-82.918,-42.601,179.092,5.831,149.308
C09794=1166.977,-83.168,-42.591,179.090,5.830,149.309
C09795=1166.982,-83.418,-42.580,179.088,5.830,149.309
C09796=1166.987,-83.667,-42.570,179.086,5.830,149.310
C09797=1166.992,-83.917,-42.560,179.083,5.829,149.311
C09798=1166.998,-84.166,-42.550,179.082,5.829,149.311
C09799=1167.003,-84.417,-42.540,179.079,5.829,149.312
C09800=1167.008,-84.666,-42.529,179.077,5.828,149.312
C09801=1167.013,-84.916,-42.521,179.075,5.828,149.313
C09802=1167.018,-85.166,-42.510,179.072,5.828,149.313
C09803=1167.024,-85.416,-42.500,179.070,5.827,149.314
C09804=1167.029,-85.665,-42.490,179.068,5.827,149.315
C09805=1167.034,-85.914,-42.480,179.066,5.826,149.315
C09806=1167.039,-86.165,-42.469,179.063,5.826,149.316
C09807=1167.045,-86.415,-42.460,179.062,5.826,149.316
C09808=1167.050,-86.664,-42.450,179.059,5.826,149.317
C09809=1167.056,-86.914,-42.440,179.057,5.826,149.318
C09810=1167.061,-87.164,-42.429,179.055,5.825,149.318
C09811=1167.066,-87.413,-42.420,179.053,5.825,149.319
C09812=1167.072,-87.663,-42.410,179.051,5.825,149.319
C09813=1167.077,-87.913,-42.400,179.048,5.824,149.320
C09814=1167.081,-88.163,-42.390,179.046,5.823,149.320
C09815=1167.087,-88.412,-42.380,179.044,5.824,149.321
C09816=1167.093,-88.662,-42.370,179.042,5.823,149.322
C09817=1167.098,-88.912,-42.361,179.039,5.823,149.322
C09818=1167.103,-89.161,-42.351,179.038,5.823,149.323
C09819=1167.108,-89.411,-42.340,179.035,5.822,149.323
C09820=1167.114,-89.661,-42.331,179.033,5.822,149.324
C09821=1167.119,-89.911,-42.321,179.031,5.821,149.324
C09822=1167.124,-90.160,-42.311,179.028,5.821,149.325
C09823=1167.130,-90.410,-42.302,179.027,5.821,149.326
C09824=1167.135,-90.661,-42.291,179.024,5.821,149.326
C09825=1167.140,-90.910,-42.282,179.022,5.820,149.327
C09826=1167.146,-91.160,-42.272,179.020,5.820,149.328
C09827=1167.151,-91.409,-42.263,179.018,5.820,149.328
C09828=1167.156,-91.659,-42.252,179.016,5.820,149.329
C09829=1167.162,-91.909,-42.243,179.013,5.819,149.329
C09830=1167.166,-92.159,-42.233,179.011,5.818,149.330
C09831=1167.172,-92.408,-42.223,179.009,5.819,149.330
C09832=1167.177,-92.658,-42.214,179.007,5.818,149.331
C09833=1167.183,-92.908,-42.204,179.005,5.818,149.332
C09834=1167.188,-93.157,-42.193,179.003,5.818,149.332
C09835=1167.193,-93.407,-42.184,179.000,5.817,149.333
C09836=1167.198,-93.657,-42.174,178.998,5.817,149.333
C09837=1167.204,-93.907,-42.165,178.996,5.817,149.334
C09838=1167.209,-94.157,-42.155,178.994,5.816,149.334
C09839=1167.214,-94.406,-42.145,178.992,5.816,149.335
C09840=1167.220,-94.656,-42.136,178.989,5.816,149.336
C09841=1167.225,-94.905,-42.126,178.988,5.816,149.336
C09842=1167.231,-95.156,-42.117,178.985,5.815,149.337
C09843=1167.236,-95.405,-42.106,178.983,5.815,149.337
C09844=1167.241,-95.656,-42.097,178.981,5.815,149.338
C09845=1167.246,-95.905,-42.087,178.979,5.814,149.339
C09846=1167.252,-96.155,-42.078,178.977,5.814,149.339
C09847=1167.257,-96.405,-42.068,178.974,5.814,149.340
C09848=1167.262,-96.654,-42.059,178.972,5.813,149.340
C09849=1167.268,-96.904,-42.049,178.970,5.814,149.341
C09850=1167.273,-97.154,-42.040,178.968,5.813,149.341
C09851=1167.279,-97.403,-42.030,178.966,5.813,149.342
C09852=1167.284,-97.653,-42.021,178.964,5.812,149.343
C09853=1167.289,-97.903,-42.010,178.962,5.812,149.343
C09854=1167.294,-98.153,-42.001,178.959,5.812,149.344
C09855=1167.300,-98.403,-41.991,178.957,5.811,149.344
C09856=1167.305,-98.653,-41.982,178.956,5.811,149.345
C09857=1167.310,-98.902,-41.972,178.953,5.811,149.346
C09858=1167.316,-99.152,-41.963,178.951,5.811,149.346
C09859=1167.321,-99.401,-41.953,178.949,5.811,149.347
C09860=1167.326,-99.652,-41.944,178.946,5.810,149.347
C09861=1167.331,-99.901,-41.934,178.945,5.810,149.348
C09862=1167.337,-100.151,-41.925,178.942,5.809,149.348
C09863=1167.342,-100.400,-41.915,178.941,5.809,149.349
C09864=1167.348,-100.650,-41.906,178.938,5.809,149.350
C09865=1167.353,-100.900,-41.897,178.936,5.808,149.350
C09866=1167.358,-101.149,-41.887,178.934,5.808,149.351
C09867=1167.364,-101.400,-41.878,178.931,5.808,149.351
C09868=1167.369,-101.649,-41.868,178.930,5.808,149.352
C09869=1167.374,-101.921,-41.858,178.927,5.808,149.352
C09870=1167.381,-102.194,-41.848,178.925,5.807,149.353
C09871=1167.386,-102.465,-41.837,178.923,5.807,149.354
C09872=1167.392,-102.737,-41.827,178.920,5.807,149.354
C09873=1167.397,-102.987,-41.818,178.918,5.806,149.355
C09874=1167.403,-103.237,-41.808,178.916,5.806,149.355
C09875=1167.408,-103.487,-41.799,178.914,5.806,149.356
C09876=1167.413,-103.736,-41.790,178.912,5.806,149.357
C09877=1167.418,-103.986,-41.780,178.909,5.805,149.357
C09878=1167.424,-104.236,-41.771,178.907,5.805,149.358
C09879=1167.428,-104.485,-41.762,178.906,5.805,149.358
C09880=1167.434,-104.735,-41.752,178.903,5.804,149.359
C09881=1167.440,-104.985,-41.743,178.901,5.804,149.359
C09882=1167.445,-105.235,-41.733,178.899,5.804,149.360
C09883=1167.450,-105.485,-41.724,178.897,5.804,149.361
C09884=1167.455,-105.734,-41.715,178.895,5.803,149.361
C09885=1167.460,-105.984,-41.706,178.893,5.804,149.362
C09886=1167.466,-106.234,-41.696,178.891,5.803,149.362
C09887=1167.471,-106.484,-41.687,178.888,5.802,149.363
C09888=1167.477,-106.733,-41.678,178.886,5.802,149.364
C09889=1167.482,-106.983,-41.668,178.884,5.802,149.364
C09890=1167.487,-107.233,-41.659,178.882,5.802,149.365
C09891=1167.493,-107.483,-41.650,178.880,5.801,149.365
C09892=1167.498,-107.733,-41.641,178.878,5.801,149.366
C09893=1167.503,-107.982,-41.631,178.876,5.801,149.366
C09894=1167.508,-108.232,-41.622,178.874,5.801,149.367
C09895=1167.514,-108.482,-41.613,178.872,5.800,149.367
C09896=1167.520,-108.731,-41.604,178.869,5.800,149.368
C09897=1167.525,-108.981,-41.595,178.868,5.800,149.369
C09898=1167.530,-109.230,-41.586,178.865,5.800,149.369
C09899=1167.535,-109.480,-41.577,178.863,5.800,149.370
C09900=1167.541,-109.730,-41.567,178.861,5.799,149.370
C09901=1167.546,-109.980,-41.559,178.859,5.799,149.371
C09902=1167.552,-110.230,-41.550,178.857,5.798,149.371
C09903=1167.557,-110.480,-41.541,178.855,5.798,149.372
C09904=1167.562,-110.729,-41.531,178.853,5.798,149.373
C09905=1167.567,-110.979,-41.522,178.850,5.797,149.373
C09906=1167.573,-111.229,-41.513,178.849,5.797,149.374
C09907=1167.578,-111.479,-41.504,178.846,5.797,149.374
C09908=1167.584,-111.729,-41.494,178.844,5.797,149.375
C09909=1167.589,-111.979,-41.485,178.842,5.796,149.375
C09910=1167.595,-112.228,-41.477,178.840,5.797,149.376
C09911=1167.600,-112.478,-41.468,178.838,5.796,149.377
C09912=1167.605,-112.727,-41.458,178.836,5.796,149.377
C09913=1167.611,-112.977,-41.449,178.834,5.796,149.378
C09914=1167.616,-113.227,-41.440,178.832,5.796,149.378
C09915=1167.621,-113.477,-41.431,178.829,5.795,149.379
C09916=1167.626,-113.727,-41.422,178.828,5.795,149.379
C09917=1167.631,-113.977,-41.413,178.826,5.794,149.380
C09918=1167.636,-114.227,-41.404,178.824,5.795,149.381
C09919=1167.643,-114.476,-41.395,178.821,5.794,149.381
C09920=1167.648,-114.726,-41.386,178.819,5.793,149.382
C09921=1167.653,-114.976,-41.377,178.817,5.794,149.382
C09922=1167.658,-115.226,-41.369,178.815,5.793,149.383
C09923=1167.664,-115.476,-41.360,178.813,5.793,149.383
C09924=1167.669,-115.725,-41.351,178.811,5.793,149.384
C09925=1167.675,-115.976,-41.341,178.809,5.793,149.384
C09926=1167.680,-116.225,-41.333,178.807,5.792,149.385
C09927=1167.686,-116.475,-41.324,178.805,5.792,149.386
C09928=1167.691,-116.724,-41.315,178.803,5.792,149.386
C09929=1167.696,-116.974,-41.306,178.801,5.792,149.387
C09930=1167.701,-117.224,-41.297,178.798,5.791,149.387
C09931=1167.706,-117.474,-41.288,178.797,5.791,149.388
C09932=1167.712,-117.723,-41.280,178.794,5.791,149.388
C09933=1167.718,-117.973,-41.270,178.793,5.791,149.389
C09934=1167.723,-118.223,-41.261,178.790,5.790,149.390
C09935=1167.728,-118.473,-41.252,178.789,5.790,149.390
C09936=1167.733,-118.723,-41.244,178.786,5.789,149.390
C09937=1167.739,-118.973,-41.235,178.784,5.790,149.391
C09938=1167.744,-119.222,-41.226,178.782,5.789,149.392
C09939=1167.750,-119.472,-41.217,178.781,5.789,149.392
C09940=1167.755,-119.722,-41.208,178.778,5.789,149.393
C09941=1167.760,-119.971,-41.199,178.776,5.789,149.393
C09942=1167.765,-120.221,-41.191,178.774,5.788,149.394
C09943=1167.770,-120.471,-41.182,178.772,5.788,149.395
C09944=1167.776,-120.721,-41.174,178.770,5.788,149.395
C09945=1167.781,-120.971,-41.165,178.768,5.788,149.396
C09946=1167.787,-121.221,-41.156,178.766,5.787,149.396
C09947=1167.792,-121.470,-41.147,178.763,5.787,149.397
C09948=1167.797,-121.720,-41.138,178.762,5.787,149.397
C09949=1167.803,-121.969,-41.130,178.760,5.786,149.398
C09950=1167.808,-122.219,-41.121,178.757,5.786,149.398
C09951=1167.813,-122.469,-41.112,178.755,5.786,149.399
C09952=1167.818,-122.720,-41.104,178.754,5.786,149.399
C09953=1167.824,-122.969,-41.095,178.751,5.785,149.400
C09954=1167.829,-123.219,-41.086,178.749,5.785,149.401
C09955=1167.835,-123.468,-41.077,178.747,5.784,149.401
C09956=1167.840,-123.718,-41.068,178.745,5.785,149.402
C09957=1167.846,-123.967,-41.060,178.743,5.784,149.402
C09958=1167.851,-124.218,-41.052,178.741,5.784,149.403
C09959=1167.856,-124.468,-41.043,178.739,5.783,149.403
C09960=1167.861,-124.718,-41.034,178.737,5.784,149.404
C09961=1167.867,-124.967,-41.025,178.735,5.784,149.404
C09962=1167.872,-125.217,-41.017,178.733,5.783,149.405
C09963=1167.878,-125.467,-41.008,178.731,5.784,149.406
C09964=1167.883,-125.717,-40.999,178.729,5.783,149.406
C09965=1167.889,-125.966,-40.991,178.727,5.783,149.407
C09966=1167.894,-126.216,-40.982,178.725,5.782,149.407
C09967=1167.899,-126.466,-40.974,178.723,5.782,149.408
C09968=1167.904,-126.716,-40.965,178.721,5.782,149.408
C09969=1167.910,-126.965,-40.956,178.719,5.782,149.409
C09970=1167.915,-127.215,-40.948,178.717,5.781,149.409
C09971=1167.921,-127.466,-40.939,178.715,5.781,149.410
C09972=1167.927,-127.715,-40.931,178.713,5.781,149.411
C09973=1167.504,-127.726,-40.972,178.709,5.784,149.412
C09974=1167.499,-127.477,-40.981,178.711,5.785,149.412
C09975=1167.495,-127.226,-40.989,178.713,5.784,149.411
C09976=1167.489,-126.977,-40.998,178.715,5.785,149.411
C09977=1167.484,-126.727,-41.006,178.717,5.785,149.410
C09978=1167.478,-126.477,-41.014,178.719,5.786,149.410
C09979=1167.473,-126.227,-41.023,178.721,5.785,149.409
C09980=1167.467,-125.978,-41.032,178.723,5.786,149.409
C09981=1167.462,-125.728,-41.041,178.725,5.786,149.408
C09982=1167.457,-125.478,-41.049,178.728,5.786,149.407
C09983=1167.451,-125.228,-41.058,178.729,5.786,149.407
C09984=1167.446,-124.979,-41.066,178.732,5.787,149.406
C09985=1167.441,-124.729,-41.075,178.733,5.787,149.406
C09986=1167.435,-124.479,-41.084,178.736,5.787,149.405
C09987=1167.430,-124.228,-41.092,178.737,5.787,149.405
C09988=1167.424,-123.979,-41.101,178.740,5.788,149.404
C09989=1167.419,-123.729,-41.110,178.741,5.788,149.404
C09990=1167.414,-123.480,-41.119,178.744,5.788,149.403
C09991=1167.409,-123.230,-41.127,178.745,5.788,149.402
C09992=1167.403,-122.980,-41.135,178.748,5.789,149.402
C09993=1167.397,-122.730,-41.144,178.750,5.789,149.401
C09994=1167.392,-122.480,-41.153,178.752,5.790,149.401
C09995=1167.387,-122.230,-41.162,178.754,5.790,149.400
C09996=1167.382,-121.981,-41.171,178.756,5.790,149.400
//INST
///DATE 2021/06/25 14:30
///ATTR SC,RW,RJ
////FRAME ROBOT
///GROUP1 RB1
NOP
MOVL C00000 V=800.0 PL=0
MOVL C00001 V=800.0 PL=0
MOVL C00002 V=800.0 PL=0
MOVL C00003 V=800.0 PL=0
MOVL C00004 V=800.0 PL=0
MOVL C00005 V=800.0 PL=0
MOVL C00006 V=800.0 PL=0
MOVL C00007 V=800.0 PL=0
MOVL C00008 V=800.0 PL=0
MOVL C00009 V=800.0 PL=0
MOVL C00010 V=800.0 PL=0
MOVL C00011 V=800.0 PL=0
MOVL C00012 V=800.0 PL=0
MOVL C00013 V=800.0 PL=0
MOVL C00014 V=800.0 PL=0
MOVL C00015 V=800.0 PL=0
MOVL C00016 V=800.0 PL=0
MOVL C00017 V=800.0 PL=0
MOVL C00018 V=800.0 PL=0
MOVL C00019 V=800.0 PL=0
MOVL C00020 V=800.0 PL=0
MOVL C00021 V=800.0 PL=0
MOVL C00022 V=800.0 PL=0
MOVL C00023 V=800.0 PL=0
MOVL C00024 V=800.0 PL=0
MOVL C00025 V=800.0 PL=0
MOVL C00026 V=800.0 PL=0
MOVL C00027 V=800.0 PL=0
MOVL C00028 V=800.0 PL=0
MOVL C00029 V=800.0 PL=0
MOVL C00030 V=800.0 PL=0
MOVL C00031 V=800.0 PL=0
MOVL C00032 V=800.0 PL=0
MOVL C00033 V=800.0 PL=0
MOVL C00034 V=800.0 PL=0
MOVL C00035 V=800.0 PL=0
MOVL C00036 V=800.0 PL=0
MOVL C00037 V=800.0 PL=0
MOVL C00038 V=800.0 PL=0
MOVL C00039 V=800.0 PL=0
MOVL C00040 V=800.0 PL=0
MOVL C00041 V=800.0 PL=0
MOVL C00042 V=800.0 PL=0
MOVL C00043 V=800.0 PL=0
MOVL C00044 V=800.0 PL=0
MOVL C00045 V=800.0 PL=0
MOVL C00046 V=800.0 PL=0
MOVL C00047 V=800.0 PL=0
MOVL C00048 V=800.0 PL=0
MOVL C00049 V=800.0 PL=0
MOVL C00050 V=800.0 PL=0
MOVL C00051 V=800.0 PL=0
MOVL C00052 V=800.0 PL=0
MOVL C00053 V=800.0 PL=0
MOVL C00054 V=800.0 PL=0
MOVL C00055 V=800.0 PL=0
MOVL C00056 V=800.0 PL=0
MOVL C00057 V=800.0 PL=0
MOVL C00058 V=800.0 PL=0
MOVL C00059 V=800.0 PL=0
MOVL C00060 V=800.0 PL=0
MOVL C00061 V=800.0 PL=0
MOVL C00062 V=800.0 PL=0
MOVL C00063 V=800.0 PL=0
MOVL C00064 V=800.0 PL=0
MOVL C00065 V=800.0 PL=0
MOVL C00066 V=800.0 PL=0
MOVL C00067 V=800.0 PL=0
MOVL C00068 V=800.0 PL=0
MOVL C00069 V=800.0 PL=0
MOVL C00070 V=800.0 PL=0
MOVL C00071 V=800.0 PL=0
MOVL C00072 V=800.0 PL=0
MOVL C00073 V=800.0 PL=0
MOVL C00074 V=800.0 PL=0
MOVL C00075 V=800.0 PL=0
MOVL C00076 V=800.0 PL=0
MOVL C00077 V=800.0 PL=0
MOVL C00078 V=800.0 PL=0
MOVL C00079 V=800.0 PL=0
MOVL C00080 V=800.0 PL=0
MOVL C00081 V=800.0 PL=0
MOVL C00082 V=800.0 PL=0
MOVL C00083 V=800.0 PL=0
MOVL C00084 V=800.0 PL=0
MOVL C00085 V=800.0 PL=0
MOVL C00086 V=800.0 PL=0
MOVL C00087 V=800.0 PL=0
MOVL C00088 V=800.0 PL=0
MOVL C00089 V=800.0 PL=0
MOVL C00090 V=800.0 PL=0
MOVL C00091 V=800.0 PL=0
MOVL C00092 V=800.0 PL=0
MOVL C00093 V=800.0 PL=0
MOVL C00094 V=800.0 PL=0
MOVL C00095 V=800.0 PL=0
MOVL C00096 V=800.0 PL=0
MOVL C00097 V=800.0 PL=0
MOVL C00098 V=800.0 PL=0
MOVL C00099 V=800.0 PL=0
MOVL C00100 V=800.0 PL=0
MOVL C00101 V=800.0 PL=0
MOVL C00102 V=800.0 PL=0
MOVL C00103 V=800.0 PL=0
MOVL C00104 V=800.0 PL=0
MOVL C00105 V=800.0 PL=0
MOVL C00106 V=800.0 PL=0
MOVL C00107 V=800.0 PL=0
MOVL C00108 V=800.0 PL=0
MOVL C00109 V=800.0 PL=0
MOVL C00110 V=800.0 PL=0
MOVL C00111 V=800.0 PL=0
MOVL C00112 V=800.0 PL=0
MOVL C00113 V=800.0 PL=0
MOVL C00114 V=800.0 PL=0
MOVL C00115 V=800.0 PL=0
MOVL C00116 V=800.0 PL=0
MOVL C00117 V=800.0 PL=0
MOVL C00118 V=800.0 PL=0
MOVL C00119 V=800.0 PL=0
MOVL C00120 V=800.0 PL=0
MOVL C00121 V=800.0 PL=0
MOVL C00122 V=800.0 PL=0
MOVL C00123 V=800.0 PL=0
MOVL C00124 V=800.0 PL=0
MOVL C00125 V=800.0 PL=0
MOVL C00126 V=800.0 PL=0
MOVL C00127 V=800.0 PL=0
MOVL C00128 V=800.0 PL=0
MOVL C00129 V=800.0 PL=0
MOVL C00130 V=800.0 PL=0
MOVL C00131 V=800.0 PL=0
MOVL C00132 V=800.0 PL=0
MOVL C00133 V=800.0 PL=0
MOVL C00134 V=800.0 PL=0
MOVL C00135 V=800.0 PL=0
MOVL C00136 V=800.0 PL=0
MOVL C00137 V=800.0 PL=0
MOVL C00138 V=800.0 PL=0
MOVL C00139 V=800.0 PL=0
MOVL C00140 V=800.0 PL=0
MOVL C00141 V=800.0 PL=0
MOVL C00142 V=800.0 PL=0
MOVL C00143 V=800.0 PL=0
MOVL C00144 V=800.0 PL=0
MOVL C00145 V=800.0 PL=0
MOVL C00146 V=800.0 PL=0
MOVL C00147 V=800.0 PL=0
MOVL C00148 V=800.0 PL=0
MOVL C00149 V=800.0 PL=0
MOVL C00150 V=800.0 PL=0
MOVL C00151 V=800.0 PL=0
MOVL C00152 V=800.0 PL=0
MOVL C00153 V=800.0 PL=0
MOVL C00154 V=800.0 PL=0
MOVL C00155 V=800.0 PL=0
MOVL C00156 V=800.0 PL=0
MOVL C00157 V=800.0 PL=0
MOVL C00158 V=800.0 PL=0
MOVL C00159 V=800.0 PL=0
MOVL C00160 V=800.0 PL=0
MOVL C00161 V=800.0 PL=0
MOVL C00162 V=800.0 PL=0
MOVL C00163 V=800.0 PL=0
MOVL C00164 V=800.0 PL=0
MOVL C00165 V=800.0 PL=0
MOVL C00166 V=800.0 PL=0
MOVL C00167 V=800.0 PL=0
MOVL C00168 V=800.0 PL=0
MOVL C00169 V=800.0 PL=0
MOVL C00170 V=800.0 PL=0
MOVL C00171 V=800.0 PL=0
MOVL C00172 V=800.0 PL=0
MOVL C00173 V=800.0 PL=0
MOVL C00174 V=800.0 PL=0
MOVL C00175 V=800.0 PL=0
MOVL C00176 V=800.0 PL=0
MOVL C00177 V=800.0 PL=0
MOVL C00178 V=800.0 PL=0
MOVL C00179 V=800.0 PL=0
MOVL C00180 V=800.0 PL=0
MOVL C00181 V=800.0 PL=0
MOVL C00182 V=800.0 PL=0
MOVL C00183 V=800.0 PL=0
MOVL C00184 V=800.0 PL=0
MOVL C00185 V=800.0 PL=0
MOVL C00186 V=800.0 PL=0
MOVL C00187 V=800.0 PL=0
MOVL C00188 V=800.0 PL=0
MOVL C00189 V=800.0 PL=0
MOVL C00190 V=800.0 PL=0
MOVL C00191 V=800.0 PL=0
MOVL C00192 V=800.0 PL=0
MOVL C00193 V=800.0 PL=0
MOVL C00194 V=800.0 PL=0
MOVL C00195 V=800.0 PL=0
MOVL C00196 V=800.0 PL=0
MOVL C00197 V=800.0 PL=0
MOVL C00198 V=800.0 PL=0
MOVL C00199 V=800.0 PL=0
MOVL C00200 V=800.0 PL=0
MOVL C00201 V=800.0 PL=0
MOVL C00202 V=800.0 PL=0
MOVL C00203 V=800.0 PL=0
MOVL C00204 V=800.0 PL=0
MOVL C00205 V=800.0 PL=0
MOVL C00206 V=800.0 PL=0
MOVL C00207 V=800.0 PL=0
MOVL C00208 V=800.0 PL=0
MOVL C00209 V=800.0 PL=0
MOVL C00210 V=800.0 PL=0
MOVL C00211 V=800.0 PL=0
MOVL C00212 V=800.0 PL=0
MOVL C00213 V=800.0 PL=0
MOVL C00214 V=800.0 PL=0
MOVL C00215 V=800.0 PL=0
MOVL C00216 V=800.0 PL=0
MOVL C00217 V=800.0 PL=0
MOVL C00218 V=800.0 PL=0
MOVL C00219 V=800.0 PL=0
MOVL C00220 V=800.0 PL=0
MOVL C00221 V=800.0 PL=0
MOVL C00222 V=800.0 PL=0
MOVL C00223 V=800.0 PL=0
MOVL C00224 V=800.0 PL=0
MOVL C00225 V=800.0 PL=0
MOVL C00226 V=800.0 PL=0
MOVL C00227 V=800.0 PL=0
MOVL C00228 V=800.0 PL=0
MOVL C00229 V=800.0 PL=0
MOVL C00230 V=800.0 PL=0
MOVL C00231 V=800.0 PL=0
MOVL C00232 V=800.0 PL=0
MOVL C00233 V=800.0 PL=0
MOVL C00234 V=800.0 PL=0
MOVL C00235 V=800.0 PL=0
MOVL C00236 V=800.0 PL=0
MOVL C00237 V=800.0 PL=0
MOVL C00238 V=800.0 PL=0
MOVL C00239 V=800.0 PL=0
MOVL C00240 V=800.0 PL=0
MOVL C00241 V=800.0 PL=0
MOVL C00242 V=800.0 PL=0
MOVL C00243 V=800.0 PL=0
MOVL C00244 V=800.0 PL=0
MOVL C00245 V=800.0 PL=0
MOVL C00246 V=800.0 PL=0
MOVL C00247 V=800.0 PL=0
MOVL C00248 V=800.0 PL=0
MOVL C00249 V=800.0 PL=0
MOVL C00250 V=800.0 PL=0
MOVL C00251 V=800.0 PL=0
MOVL C00252 V=800.0 PL=0
MOVL C00253 V=800.0 PL=0
MOVL C00254 V=800.0 PL=0
MOVL C00255 V=800.0 PL=0
MOVL C00256 V=800.0 PL=0
MOVL C00257 V=800.0 PL=0
MOVL C00258 V=800.0 PL=0
MOVL C00259 V=800.0 PL=0
MOVL C00260 V=800.0 PL=0
MOVL C00261 V=800.0 PL=0
MOVL C00262 V=800.0 PL=0
MOVL C00263 V=800.0 PL=0
MOVL C00264 V=800.0 PL=0
MOVL C00265 V=800.0 PL=0
MOVL C00266 V=800.0 PL=0
MOVL C00267 V=800.0 PL=0
MOVL C00268 V=800.0 PL=0
MOVL C00269 V=800.0 PL=0
MOVL C00270 V=800.0 PL=0
MOVL C00271 V=800.0 PL=0
MOVL C00272 V=800.0 PL=0
MOVL C00273 V=800.0 PL=0
MOVL C00274 V=800.0 PL=0
MOVL C00275 V=800.0 PL=0
MOVL C00276 V=800.0 PL=0
MOVL C00277 V=800.0 PL=0
MOVL C00278 V=800.0 PL=0
MOVL C00279 V=800.0 PL=0
MOVL C00280 V=800.0 PL=0
MOVL C00281 V=800.0 PL=0
MOVL C00282 V=800.0 PL=0
MOVL C00283 V=800.0 PL=0
MOVL C00284 V=800.0 PL=0
MOVL C00285 V=800.0 PL=0
MOVL C00286 V=800.0 PL=0
MOVL C00287 V=800.0 PL=0
MOVL C00288 V=800.0 PL=0
MOVL C00289 V=800.0 PL=0
MOVL C00290 V=800.0 PL=0
MOVL C00291 V=800.0 PL=0
MOVL C00292 V=800.0 PL=0
MOVL C00293 V=800.0 PL=0
MOVL C00294 V=800.0 PL=0
MOVL C00295 V=800.0 PL=0
MOVL C00296 V=800.0 PL=0
MOVL C00297 V=800.0 PL=0
MOVL C00298 V=800.0 PL=0
MOVL C00299 V=800.0 PL=0
MOVL C00300 V=800.0 PL=0
MOVL C00301 V=800.0 PL=0
MOVL C00302 V=800.0 PL=0
MOVL C00303 V=800.0 PL=0
MOVL C00304 V=800.0 PL=0
MOVL C00305 V=800.0 PL=0
MOVL C00306 V=800.0 PL=0
MOVL C00307 V=800.0 PL=0
MOVL C00308 V=800.0 PL=0
MOVL C00309 V=800.0 PL=0
MOVL C00310 V=800.0 PL=0
MOVL C00311 V=800.0 PL=0
MOVL C00312 V=800.0 PL=0
MOVL C00313 V=800.0 PL=0
MOVL C00314 V=800.0 PL=0
MOVL C00315 V=800.0 PL=0
MOVL C00316 V=800.0 PL=0
MOVL C00317 V=800.0 PL=0
MOVL C00318 V=800.0 PL=0
MOVL C00319 V=800.0 PL=0
MOVL C00320 V=800.0 PL=0
MOVL C00321 V=800.0 PL=0
MOVL C00322 V=800.0 PL=0
MOVL C00323 V=800.0 PL=0
MOVL C00324 V=800.0 PL=0
MOVL C00325 V=800.0 PL=0
MOVL C00326 V=800.0 PL=0
MOVL C00327 V=800.0 PL=0
MOVL C00328 V=800.0 PL=0
MOVL C00329 V=800.0 PL=0
MOVL C00330 V=800.0 PL=0
MOVL C00331 V=800.0 PL=0
MOVL C00332 V=800.0 PL=0
MOVL C00333 V=800.0 PL=0
MOVL C00334 V=800.0 PL=0
MOVL C00335 V=800.0 PL=0
MOVL C00336 V=800.0 PL=0
MOVL C00337 V=800.0 PL=0
MOVL C00338 V=800.0 PL=0
MOVL C00339 V=800.0 PL=0
MOVL C00340 V=800.0 PL=0
MOVL C00341 V=800.0 PL=0
MOVL C00342 V=800.0 PL=0
MOVL C00343 V=800.0 PL=0
MOVL C00344 V=800.0 PL=0
MOVL C00345 V=800.0 PL=0
MOVL C00346 V=800.0 PL=0
MOVL C00347 V=800.0 PL=0
MOVL C00348 V=800.0 PL=0
MOVL C00349 V=800.0 PL=0
MOVL C00350 V=800.0 PL=0
MOVL C00351 V=800.0 PL=0
MOVL C00352 V=800.0 PL=0
MOVL C00353 V=800.0 PL=0
MOVL C00354 V=800.0 PL=0
MOVL C00355 V=800.0 PL=0
MOVL C00356 V=800.0 PL=0
MOVL C00357 V=800.0 PL=0
MOVL C00358 V=800.0 PL=0
MOVL C00359 V=800.0 PL=0
MOVL C00360 V=800.0 PL=0
MOVL C00361 V=800.0 PL=0
MOVL C00362 V=800.0 PL=0
MOVL C00363 V=800.0 PL=0
MOVL C00364 V=800.0 PL=0
MOVL C00365 V=800.0 PL=0
MOVL C00366 V=800.0 PL=0
MOVL C00367 V=800.0 PL=0
MOVL C00368 V=800.0 PL=0
MOVL C00369 V=800.0 PL=0
MOVL C00370 V=800.0 PL=0
MOVL C00371 V=800.0 PL=0
MOVL C00372 V=800.0 PL=0
MOVL C00373 V=800.0 PL=0
MOVL C00374 V=800.0 PL=0
MOVL C00375 V=800.0 PL=0
MOVL C00376 V=800.0 PL=0
MOVL C00377 V=800.0 PL=0
MOVL C00378 V=800.0 PL=0
MOVL C00379 V=800.0 PL=0
MOVL C00380 V=800.0 PL=0
MOVL C00381 V=800.0 PL=0
MOVL C00382 V=800.0 PL=0
MOVL C00383 V=800.0 PL=0
MOVL C00384 V=800.0 PL=0
MOVL C00385 V=800.0 PL=0
MOVL C00386 V=800.0 PL=0
MOVL C00387 V=800.0 PL=0
MOVL C00388 V=800.0 PL=0
MOVL C00389 V=800.0 PL=0
MOVL C00390 V=800.0 PL=0
MOVL C00391 V=800.0 PL=0
MOVL C00392 V=800.0 PL=0
MOVL C00393 V=800.0 PL=0
MOVL C00394 V=800.0 PL=0
MOVL C00395 V=800.0 PL=0
MOVL C00396 V=800.0 PL=0
MOVL C00397 V=800.0 PL=0
MOVL C00398 V=800.0 PL=0
MOVL C00399 V=800.0 PL=0
MOVL C00400 V=800.0 PL=0
MOVL C00401 V=800.0 PL=0
MOVL C00402 V=800.0 PL=0
MOVL C00403 V=800.0 PL=0
MOVL C00404 V=800.0 PL=0
MOVL C00405 V=800.0 PL=0
MOVL C00406 V=800.0 PL=0
MOVL C00407 V=800.0 PL=0
MOVL C00408 V=800.0 PL=0
MOVL C00409 V=800.0 PL=0
MOVL C00410 V=800.0 PL=0
MOVL C00411 V=800.0 PL=0
MOVL C00412 V=800.0 PL=0
MOVL C00413 V=800.0 PL=0
MOVL C00414 V=800.0 PL=0
MOVL C00415 V=800.0 PL=0
MOVL C00416 V=800.0 PL=0
MOVL C00417 V=800.0 PL=0
MOVL C00418 V=800.0 PL=0
MOVL C00419 V=800.0 PL=0
MOVL C00420 V=800.0 PL=0
MOVL C00421 V=800.0 PL=0
MOVL C00422 V=800.0 PL=0
MOVL C00423 V=800.0 PL=0
MOVL C00424 V=800.0 PL=0
MOVL C00425 V=800.0 PL=0
MOVL C00426 V=800.0 PL=0
MOVL C00427 V=800.0 PL=0
MOVL C00428 V=800.0 PL=0
MOVL C00429 V=800.0 PL=0
MOVL C00430 V=800.0 PL=0
MOVL C00431 V=800.0 PL=0
MOVL C00432 V=800.0 PL=0
MOVL C00433 V=800.0 PL=0
MOVL C00434 V=800.0 PL=0
MOVL C00435 V=800.0 PL=0
MOVL C00436 V=800.0 PL=0
MOVL C00437 V=800.0 PL=0
MOVL C00438 V=800.0 PL=0
MOVL C00439 V=800.0 PL=0
MOVL C00440 V=800.0 PL=0
MOVL C00441 V=800.0 PL=0
MOVL C00442 V=800.0 PL=0
MOVL C00443 V=800.0 PL=0
MOVL C00444 V=800.0 PL=0
MOVL C00445 V=800.0 PL=0
MOVL C00446 V=800.0 PL=0
MOVL C00447 V=800.0 PL=0
MOVL C00448 V=800.0 PL=0
MOVL C00449 V=800.0 PL=0
MOVL C00450 V=800.0 PL=0
MOVL C00451 V=800.0 PL=0
MOVL C00452 V=800.0 PL=0
MOVL C00453 V=800.0 PL=0
MOVL C00454 V=800.0 PL=0
MOVL C00455 V=800.0 PL=0
MOVL C00456 V=800.0 PL=0
MOVL C00457 V=800.0 PL=0
MOVL C00458 V=800.0 PL=0
MOVL C00459 V=800.0 PL=0
MOVL C00460 V=800.0 PL=0
MOVL C00461 V=800.0 PL=0
MOVL C00462 V=800.0 PL=0
MOVL C00463 V=800.0 PL=0
MOVL C00464 V=800.0 PL=0
MOVL C00465 V=800.0 PL=0
MOVL C00466 V=800.0 PL=0
MOVL C00467 V=800.0 PL=0
MOVL C00468 V=800.0 PL=0
MOVL C00469 V=800.0 PL=0
MOVL C00470 V=800.0 PL=0
MOVL C00471 V=800.0 PL=0
MOVL C00472 V=800.0 PL=0
MOVL C00473 V=800.0 PL=0
MOVL C00474 V=800.0 PL=0
MOVL C00475 V=800.0 PL=0
MOVL C00476 V=800.0 PL=0
MOVL C00477 V=800.0 PL=0
MOVL C00478 V=800.0 PL=0
MOVL C00479 V=800.0 PL=0
MOVL C00480 V=800.0 PL=0
MOVL C00481 V=800.0 PL=0
MOVL C00482 V=800.0 PL=0
MOVL C00483 V=800.0 PL=0
MOVL C00484 V=800.0 PL=0
MOVL C00485 V=800.0 PL=0
MOVL C00486 V=800.0 PL=0
MOVL C00487 V=800.0 PL=0
MOVL C00488 V=800.0 PL=0
MOVL C00489 V=800.0 PL=0
MOVL C00490 V=800.0 PL=0
MOVL C00491 V=800.0 PL=0
MOVL C00492 V=800.0 PL=0
MOVL C00493 V=800.0 PL=0
MOVL C00494 V=800.0 PL=0
MOVL C00495 V=800.0 PL=0
MOVL C00496 V=800.0 PL=0
MOVL C00497 V=800.0 PL=0
MOVL C00498 V=800.0 PL=0
MOVL C00499 V=800.0 PL=0
MOVL C00500 V=800.0 PL=0
MOVL C00501 V=800.0 PL=0
MOVL C00502 V=800.0 PL=0
MOVL C00503 V=800.0 PL=0
MOVL C00504 V=800.0 PL=0
MOVL C00505 V=800.0 PL=0
MOVL C00506 V=800.0 PL=0
MOVL C00507 V=800.0 PL=0
MOVL C00508 V=800.0 PL=0
MOVL C00509 V=800.0 PL=0
MOVL C00510 V=800.0 PL=0
MOVL C00511 V=800.0 PL=0
MOVL C00512 V=800.0 PL=0
MOVL C00513 V=800.0 PL=0
MOVL C00514 V=800.0 PL=0
MOVL C00515 V=800.0 PL=0
MOVL C00516 V=800.0 PL=0
MOVL C00517 V=800.0 PL=0
MOVL C00518 V=800.0 PL=0
MOVL C00519 V=800.0 PL=0
MOVL C00520 V=800.0 PL=0
MOVL C00521 V=800.0 PL=0
MOVL C00522 V=800.0 PL=0
MOVL C00523 V=800.0 PL=0
MOVL C00524 V=800.0 PL=0
MOVL C00525 V=800.0 PL=0
MOVL C00526 V=800.0 PL=0
MOVL C00527 V=800.0 PL=0
MOVL C00528 V=800.0 PL=0
MOVL C00529 V=800.0 PL=0
MOVL C00530 V=800.0 PL=0
MOVL C00531 V=800.0 PL=0
MOVL C00532 V=800.0 PL=0
MOVL C00533 V=800.0 PL=0
MOVL C00534 V=800.0 PL=0
MOVL C00535 V=800.0 PL=0
MOVL C00536 V=800.0 PL=0
MOVL C00537 V=800.0 PL=0
MOVL C00538 V=800.0 PL=0
MOVL C00539 V=800.0 PL=0
MOVL C00540 V=800.0 PL=0
MOVL C00541 V=800.0 PL=0
MOVL C00542 V=800.0 PL=0
MOVL C00543 V=800.0 PL=0
MOVL C00544 V=800.0 PL=0
MOVL C00545 V=800.0 PL=0
MOVL C00546 V=800.0 PL=0
MOVL C00547 V=800.0 PL=0
MOVL C00548 V=800.0 PL=0
MOVL C00549 V=800.0 PL=0
MOVL C00550 V=800.0 PL=0
MOVL C00551 V=800.0 PL=0
MOVL C00552 V=800.0 PL=0
MOVL C00553 V=800.0 PL=0
MOVL C00554 V=800.0 PL=0
MOVL C00555 V=800.0 PL=0
MOVL C00556 V=800.0 PL=0
MOVL C00557 V=800.0 PL=0
MOVL C00558 V=800.0 PL=0
MOVL C00559 V=800.0 PL=0
MOVL C00560 V=800.0 PL=0
MOVL C00561 V=800.0 PL=0
MOVL C00562 V=800.0 PL=0
MOVL C00563 V=800.0 PL=0
MOVL C00564 V=800.0 PL=0
MOVL C00565 V=800.0 PL=0
MOVL C00566 V=800.0 PL=0
MOVL C00567 V=800.0 PL=0
MOVL C00568 V=800.0 PL=0
MOVL C00569 V=800.0 PL=0
MOVL C00570 V=800.0 PL=0
MOVL C00571 V=800.0 PL=0
MOVL C00572 V=800.0 PL=0
MOVL C00573 V=800.0 PL=0
MOVL C00574 V=800.0 PL=0
MOVL C00575 V=800.0 PL=0
MOVL C00576 V=800.0 PL=0
MOVL C00577 V=800.0 PL=0
MOVL C00578 V=800.0 PL=0
MOVL C00579 V=800.0 PL=0
MOVL C00580 V=800.0 PL=0
MOVL C00581 V=800.0 PL=0
MOVL C00582 V=800.0 PL=0
MOVL C00583 V=800.0 PL=0
MOVL C00584 V=800.0 PL=0
MOVL C00585 V=800.0 PL=0
MOVL C00586 V=800.0 PL=0
MOVL C00587 V=800.0 PL=0
MOVL C00588 V=800.0 PL=0
MOVL C00589 V=800.0 PL=0
MOVL C00590 V=800.0 PL=0
MOVL C00591 V=800.0 PL=0
MOVL C00592 V=800.0 PL=0
MOVL C00593 V=800.0 PL=0
MOVL C00594 V=800.0 PL=0
MOVL C00595 V=800.0 PL=0
MOVL C00596 V=800.0 PL=0
MOVL C00597 V=800.0 PL=0
MOVL C00598 V=800.0 PL=0
MOVL C00599 V=800.0 PL=0
MOVL C00600 V=800.0 PL=0
MOVL C00601 V=800.0 PL=0
MOVL C00602 V=800.0 PL=0
MOVL C00603 V=800.0 PL=0
MOVL C00604 V=800.0 PL=0
MOVL C00605 V=800.0 PL=0
MOVL C00606 V=800.0 PL=0
MOVL C00607 V=800.0 PL=0
MOVL C00608 V=800.0 PL=0
MOVL C00609 V=800.0 PL=0
MOVL C00610 V=800.0 PL=0
MOVL C00611 V=800.0 PL=0
MOVL C00612 V=800.0 PL=0
MOVL C00613 V=800.0 PL=0
MOVL C00614 V=800.0 PL=0
MOVL C00615 V=800.0 PL=0
MOVL C00616 V=800.0 PL=0
MOVL C00617 V=800.0 PL=0
MOVL C00618 V=800.0 PL=0
MOVL C00619 V=800.0 PL=0
MOVL C00620 V=800.0 PL=0
MOVL C00621 V=800.0 PL=0
MOVL C00622 V=800.0 PL=0
MOVL C00623 V=800.0 PL=0
MOVL C00624 V=800.0 PL=0
MOVL C00625 V=800.0 PL=0
MOVL C00626 V=800.0 PL=0
MOVL C00627 V=800.0 PL=0
MOVL C00628 V=800.0 PL=0
MOVL C00629 V=800.0 PL=0
MOVL C00630 V=800.0 PL=0
MOVL C00631 V=800.0 PL=0
MOVL C00632 V=800.0 PL=0
MOVL C00633 V=800.0 PL=0
MOVL C00634 V=800.0 PL=0
MOVL C00635 V=800.0 PL=0
MOVL C00636 V=800.0 PL=0
MOVL C00637 V=800.0 PL=0
MOVL C00638 V=800.0 PL=0
MOVL C00639 V=800.0 PL=0
MOVL C00640 V=800.0 PL=0
MOVL C00641 V=800.0 PL=0
MOVL C00642 V=800.0 PL=0
MOVL C00643 V=800.0 PL=0
MOVL C00644 V=800.0 PL=0
MOVL C00645 V=800.0 PL=0
MOVL C00646 V=800.0 PL=0
MOVL C00647 V=800.0 PL=0
MOVL C00648 V=800.0 PL=0
MOVL C00649 V=800.0 PL=0
MOVL C00650 V=800.0 PL=0
MOVL C00651 V=800.0 PL=0
MOVL C00652 V=800.0 PL=0
MOVL C00653 V=800.0 PL=0
MOVL C00654 V=800.0 PL=0
MOVL C00655 V=800.0 PL=0
MOVL C00656 V=800.0 PL=0
MOVL C00657 V=800.0 PL=0
MOVL C00658 V=800.0 PL=0
MOVL C00659 V=800.0 PL=0
MOVL C00660 V=800.0 PL=0
MOVL C00661 V=800.0 PL=0
MOVL C00662 V=800.0 PL=0
MOVL C00663 V=800.0 PL=0
MOVL C00664 V=800.0 PL=0
MOVL C00665 V=800.0 PL=0
MOVL C00666 V=800.0 PL=0
MOVL C00667 V=800.0 PL=0
MOVL C00668 V=800.0 PL=0
MOVL C00669 V=800.0 PL=0
MOVL C00670 V=800.0 PL=0
MOVL C00671 V=800.0 PL=0
MOVL C00672 V=800.0 PL=0
MOVL C00673 V=800.0 PL=0
MOVL C00674 V=800.0 PL=0
MOVL C00675 V=800.0 PL=0
MOVL C00676 V=800.0 PL=0
MOVL C00677 V=800.0 PL=0
MOVL C00678 V=800.0 PL=0
MOVL C00679 V=800.0 PL=0
MOVL C00680 V=800.0 PL=0
MOVL C00681 V=800.0 PL=0
MOVL C00682 V=800.0 PL=0
MOVL C00683 V=800.0 PL=0
MOVL C00684 V=800.0 PL=0
MOVL C00685 V=800.0 PL=0
MOVL C00686 V=800.0 PL=0
MOVL C00687 V=800.0 PL=0
MOVL C00688 V=800.0 PL=0
MOVL C00689 V=800.0 PL=0
MOVL C00690 V=800.0 PL=0
MOVL C00691 V=800.0 PL=0
MOVL C00692 V=800.0 PL=0
MOVL C00693 V=800.0 PL=0
MOVL C00694 V=800.0 PL=0
MOVL C00695 V=800.0 PL=0
MOVL C00696 V=800.0 PL=0
MOVL C00697 V=800.0 PL=0
MOVL C00698 V=800.0 PL=0
MOVL C00699 V=800.0 PL=0
MOVL C00700 V=800.0 PL=0
MOVL C00701 V=800.0 PL=0
MOVL C00702 V=800.0 PL=0
MOVL C00703 V=800.0 PL=0
MOVL C00704 V=800.0 PL=0
MOVL C00705 V=800.0 PL=0
MOVL C00706 V=800.0 PL=0
MOVL C00707 V=800.0 PL=0
MOVL C00708 V=800.0 PL=0
MOVL C00709 V=800.0 PL=0
MOVL C00710 V=800.0 PL=0
MOVL C00711 V=800.0 PL=0
MOVL C00712 V=800.0 PL=0
MOVL C00713 V=800.0 PL=0
MOVL C00714 V=800.0 PL=0
MOVL C00715 V=800.0 PL=0
MOVL C00716 V=800.0 PL=0
MOVL C00717 V=800.0 PL=0
MOVL C00718 V=800.0 PL=0
MOVL C00719 V=800.0 PL=0
MOVL C00720 V=800.0 PL=0
MOVL C00721 V=800.0 PL=0
MOVL C00722 V=800.0 PL=0
MOVL C00723 V=800.0 PL=0
MOVL C00724 V=800.0 PL=0
MOVL C00725 V=800.0 PL=0
MOVL C00726 V=800.0 PL=0
MOVL C00727 V=800.0 PL=0
MOVL C00728 V=800.0 PL=0
MOVL C00729 V=800.0 PL=0
MOVL C00730 V=800.0 PL=0
MOVL C00731 V=800.0 PL=0
MOVL C00732 V=800.0 PL=0
MOVL C00733 V=800.0 PL=0
MOVL C00734 V=800.0 PL=0
MOVL C00735 V=800.0 PL=0
MOVL C00736 V=800.0 PL=0
MOVL C00737 V=800.0 PL=0
MOVL C00738 V=800.0 PL=0
MOVL C00739 V=800.0 PL=0
MOVL C00740 V=800.0 PL=0
MOVL C00741 V=800.0 PL=0
MOVL C00742 V=800.0 PL=0
MOVL C00743 V=800.0 PL=0
MOVL C00744 V=800.0 PL=0
MOVL C00745 V=800.0 PL=0
MOVL C00746 V=800.0 PL=0
MOVL C00747 V=800.0 PL=0
MOVL C00748 V=800.0 PL=0
MOVL C00749 V=800.0 PL=0
MOVL C00750 V=800.0 PL=0
MOVL C00751 V=800.0 PL=0
MOVL C00752 V=800.0 PL=0
MOVL C00753 V=800.0 PL=0
MOVL C00754 V=800.0 PL=0
MOVL C00755 V=800.0 PL=0
MOVL C00756 V=800.0 PL=0
MOVL C00757 V=800.0 PL=0
MOVL C00758 V=800.0 PL=0
MOVL C00759 V=800.0 PL=0
MOVL C00760 V=800.0 PL=0
MOVL C00761 V=800.0 PL=0
MOVL C00762 V=800.0 PL=0
MOVL C00763 V=800.0 PL=0
MOVL C00764 V=800.0 PL=0
MOVL C00765 V=800.0 PL=0
MOVL C00766 V=800.0 PL=0
MOVL C00767 V=800.0 PL=0
MOVL C00768 V=800.0 PL=0
MOVL C00769 V=800.0 PL=0
MOVL C00770 V=800.0 PL=0
MOVL C00771 V=800.0 PL=0
MOVL C00772 V=800.0 PL=0
MOVL C00773 V=800.0 PL=0
MOVL C00774 V=800.0 PL=0
MOVL C00775 V=800.0 PL=0
MOVL C00776 V=800.0 PL=0
MOVL C00777 V=800.0 PL=0
MOVL C00778 V=800.0 PL=0
MOVL C00779 V=800.0 PL=0
MOVL C00780 V=800.0 PL=0
MOVL C00781 V=800.0 PL=0
MOVL C00782 V=800.0 PL=0
MOVL C00783 V=800.0 PL=0
MOVL C00784 V=800.0 PL=0
MOVL C00785 V=800.0 PL=0
MOVL C00786 V=800.0 PL=0
MOVL C00787 V=800.0 PL=0
MOVL C00788 V=800.0 PL=0
MOVL C00789 V=800.0 PL=0
MOVL C00790 V=800.0 PL=0
MOVL C00791 V=800.0 PL=0
MOVL C00792 V=800.0 PL=0
MOVL C00793 V=800.0 PL=0
MOVL C00794 V=800.0 PL=0
MOVL C00795 V=800.0 PL=0
MOVL C00796 V=800.0 PL=0
MOVL C00797 V=800.0 PL=0
MOVL C00798 V=800.0 PL=0
MOVL C00799 V=800.0 PL=0
MOVL C00800 V=800.0 PL=0
MOVL C00801 V=800.0 PL=0
MOVL C00802 V=800.0 PL=0
MOVL C00803 V=800.0 PL=0
MOVL C00804 V=800.0 PL=0
MOVL C00805 V=800.0 PL=0
MOVL C00806 V=800.0 PL=0
MOVL C00807 V=800.0 PL=0
MOVL C00808 V=800.0 PL=0
MOVL C00809 V=800.0 PL=0
MOVL C00810 V=800.0 PL=0
MOVL C00811 V=800.0 PL=0
MOVL C00812 V=800.0 PL=0
MOVL C00813 V=800.0 PL=0
MOVL C00814 V=800.0 PL=0
MOVL C00815 V=800.0 PL=0
MOVL C00816 V=800.0 PL=0
MOVL C00817 V=800.0 PL=0
MOVL C00818 V=800.0 PL=0
MOVL C00819 V=800.0 PL=0
MOVL C00820 V=800.0 PL=0
MOVL C00821 V=800.0 PL=0
MOVL C00822 V=800.0 PL=0
MOVL C00823 V=800.0 PL=0
MOVL C00824 V=800.0 PL=0
MOVL C00825 V=800.0 PL=0
MOVL C00826 V=800.0 PL=0
MOVL C00827 V=800.0 PL=0
MOVL C00828 V=800.0 PL=0
MOVL C00829 V=800.0 PL=0
MOVL C00830 V=800.0 PL=0
MOVL C00831 V=800.0 PL=0
MOVL C00832 V=800.0 PL=0
MOVL C00833 V=800.0 PL=0
MOVL C00834 V=800.0 PL=0
MOVL C00835 V=800.0 PL=0
MOVL C00836 V=800.0 PL=0
MOVL C00837 V=800.0 PL=0
MOVL C00838 V=800.0 PL=0
MOVL C00839 V=800.0 PL=0
MOVL C00840 V=800.0 PL=0
MOVL C00841 V=800.0 PL=0
MOVL C00842 V=800.0 PL=0
MOVL C00843 V=800.0 PL=0
MOVL C00844 V=800.0 PL=0
MOVL C00845 V=800.0 PL=0
MOVL C00846 V=800.0 PL=0
MOVL C00847 V=800.0 PL=0
MOVL C00848 V=800.0 PL=0
MOVL C00849 V=800.0 PL=0
MOVL C00850 V=800.0 PL=0
MOVL C00851 V=800.0 PL=0
MOVL C00852 V=800.0 PL=0
MOVL C00853 V=800.0 PL=0
MOVL C00854 V=800.0 PL=0
MOVL C00855 V=800.0 PL=0
MOVL C00856 V=800.0 PL=0
MOVL C00857 V=800.0 PL=0
MOVL C00858 V=800.0 PL=0
MOVL C00859 V=800.0 PL=0
MOVL C00860 V=800.0 PL=0
MOVL C00861 V=800.0 PL=0
MOVL C00862 V=800.0 PL=0
MOVL C00863 V=800.0 PL=0
MOVL C00864 V=800.0 PL=0
MOVL C00865 V=800.0 PL=0
MOVL C00866 V=800.0 PL=0
MOVL C00867 V=800.0 PL=0
MOVL C00868 V=800.0 PL=0
MOVL C00869 V=800.0 PL=0
MOVL C00870 V=800.0 PL=0
MOVL C00871 V=800.0 PL=0
MOVL C00872 V=800.0 PL=0
MOVL C00873 V=800.0 PL=0
MOVL C00874 V=800.0 PL=0
MOVL C00875 V=800.0 PL=0
MOVL C00876 V=800.0 PL=0
MOVL C00877 V=800.0 PL=0
MOVL C00878 V=800.0 PL=0
MOVL C00879 V=800.0 PL=0
MOVL C00880 V=800.0 PL=0
MOVL C00881 V=800.0 PL=0
MOVL C00882 V=800.0 PL=0
MOVL C00883 V=800.0 PL=0
MOVL C00884 V=800.0 PL=0
MOVL C00885 V=800.0 PL=0
MOVL C00886 V=800.0 PL=0
MOVL C00887 V=800.0 PL=0
MOVL C00888 V=800.0 PL=0
MOVL C00889 V=800.0 PL=0
MOVL C00890 V=800.0 PL=0
MOVL C00891 V=800.0 PL=0
MOVL C00892 V=800.0 PL=0
MOVL C00893 V=800.0 PL=0
MOVL C00894 V=800.0 PL=0
MOVL C00895 V=800.0 PL=0
MOVL C00896 V=800.0 PL=0
MOVL C00897 V=800.0 PL=0
MOVL C00898 V=800.0 PL=0
MOVL C00899 V=800.0 PL=0
MOVL C00900 V=800.0 PL=0
MOVL C00901 V=800.0 PL=0
MOVL C00902 V=800.0 PL=0
MOVL C00903 V=800.0 PL=0
MOVL C00904 V=800.0 PL=0
MOVL C00905 V=800.0 PL=0
MOVL C00906 V=800.0 PL=0
MOVL C00907 V=800.0 PL=0
MOVL C00908 V=800.0 PL=0
MOVL C00909 V=800.0 PL=0
MOVL C00910 V=800.0 PL=0
MOVL C00911 V=800.0 PL=0
MOVL C00912 V=800.0 PL=0
MOVL C00913 V=800.0 PL=0
MOVL C00914 V=800.0 PL=0
MOVL C00915 V=800.0 PL=0
MOVL C00916 V=800.0 PL=0
MOVL C00917 V=800.0 PL=0
MOVL C00918 V=800.0 PL=0
MOVL C00919 V=800.0 PL=0
MOVL C00920 V=800.0 PL=0
MOVL C00921 V=800.0 PL=0
MOVL C00922 V=800.0 PL=0
MOVL C00923 V=800.0 PL=0
MOVL C00924 V=800.0 PL=0
MOVL C00925 V=800.0 PL=0
MOVL C00926 V=800.0 PL=0
MOVL C00927 V=800.0 PL=0
MOVL C00928 V=800.0 PL=0
MOVL C00929 V=800.0 PL=0
MOVL C00930 V=800.0 PL=0
MOVL C00931 V=800.0 PL=0
MOVL C00932 V=800.0 PL=0
MOVL C00933 V=800.0 PL=0
MOVL C00934 V=800.0 PL=0
MOVL C00935 V=800.0 PL=0
MOVL C00936 V=800.0 PL=0
MOVL C00937 V=800.0 PL=0
MOVL C00938 V=800.0 PL=0
MOVL C00939 V=800.0 PL=0
MOVL C00940 V=800.0 PL=0
MOVL C00941 V=800.0 PL=0
MOVL C00942 V=800.0 PL=0
MOVL C00943 V=800.0 PL=0
MOVL C00944 V=800.0 PL=0
MOVL C00945 V=800.0 PL=0
MOVL C00946 V=800.0 PL=0
MOVL C00947 V=800.0 PL=0
MOVL C00948 V=800.0 PL=0
MOVL C00949 V=800.0 PL=0
MOVL C00950 V=800.0 PL=0
MOVL C00951 V=800.0 PL=0
MOVL C00952 V=800.0 PL=0
MOVL C00953 V=800.0 PL=0
MOVL C00954 V=800.0 PL=0
MOVL C00955 V=800.0 PL=0
MOVL C00956 V=800.0 PL=0
MOVL C00957 V=800.0 PL=0
MOVL C00958 V=800.0 PL=0
MOVL C00959 V=800.0 PL=0
MOVL C00960 V=800.0 PL=0
MOVL C00961 V=800.0 PL=0
MOVL C00962 V=800.0 PL=0
MOVL C00963 V=800.0 PL=0
MOVL C00964 V=800.0 PL=0
MOVL C00965 V=800.0 PL=0
MOVL C00966 V=800.0 PL=0
MOVL C00967 V=800.0 PL=0
MOVL C00968 V=800.0 PL=0
MOVL C00969 V=800.0 PL=0
MOVL C00970 V=800.0 PL=0
MOVL C00971 V=800.0 PL=0
MOVL C00972 V=800.0 PL=0
MOVL C00973 V=800.0 PL=0
MOVL C00974 V=800.0 PL=0
MOVL C00975 V=800.0 PL=0
MOVL C00976 V=800.0 PL=0
MOVL C00977 V=800.0 PL=0
MOVL C00978 V=800.0 PL=0
MOVL C00979 V=800.0 PL=0
MOVL C00980 V=800.0 PL=0
MOVL C00981 V=800.0 PL=0
MOVL C00982 V=800.0 PL=0
MOVL C00983 V=800.0 PL=0
MOVL C00984 V=800.0 PL=0
MOVL C00985 V=800.0 PL=0
MOVL C00986 V=800.0 PL=0
MOVL C00987 V=800.0 PL=0
MOVL C00988 V=800.0 PL=0
MOVL C00989 V=800.0 PL=0
MOVL C00990 V=800.0 PL=0
MOVL C00991 V=800.0 PL=0
MOVL C00992 V=800.0 PL=0
MOVL C00993 V=800.0 PL=0
MOVL C00994 V=800.0 PL=0
MOVL C00995 V=800.0 PL=0
MOVL C00996 V=800.0 PL=0
MOVL C00997 V=800.0 PL=0
MOVL C00998 V=800.0 PL=0
MOVL C00999 V=800.0 PL=0
MOVL C01000 V=800.0 PL=0
MOVL C01001 V=800.0 PL=0
MOVL C01002 V=800.0 PL=0
MOVL C01003 V=800.0 PL=0
MOVL C01004 V=800.0 PL=0
MOVL C01005 V=800.0 PL=0
MOVL C01006 V=800.0 PL=0
MOVL C01007 V=800.0 PL=0
MOVL C01008 V=800.0 PL=0
MOVL C01009 V=800.0 PL=0
MOVL C01010 V=800.0 PL=0
MOVL C01011 V=800.0 PL=0
MOVL C01012 V=800.0 PL=0
MOVL C01013 V=800.0 PL=0
MOVL C01014 V=800.0 PL=0
MOVL C01015 V=800.0 PL=0
MOVL C01016 V=800.0 PL=0
MOVL C01017 V=800.0 PL=0
MOVL C01018 V=800.0 PL=0
MOVL C01019 V=800.0 PL=0
MOVL C01020 V=800.0 PL=0
MOVL C01021 V=800.0 PL=0
MOVL C01022 V=800.0 PL=0
MOVL C01023 V=800.0 PL=0
MOVL C01024 V=800.0 PL=0
MOVL C01025 V=800.0 PL=0
MOVL C01026 V=800.0 PL=0
MOVL C01027 V=800.0 PL=0
MOVL C01028 V=800.0 PL=0
MOVL C01029 V=800.0 PL=0
MOVL C01030 V=800.0 PL=0
MOVL C01031 V=800.0 PL=0
MOVL C01032 V=800.0 PL=0
MOVL C01033 V=800.0 PL=0
MOVL C01034 V=800.0 PL=0
MOVL C01035 V=800.0 PL=0
MOVL C01036 V=800.0 PL=0
MOVL C01037 V=800.0 PL=0
MOVL C01038 V=800.0 PL=0
MOVL C01039 V=800.0 PL=0
MOVL C01040 V=800.0 PL=0
MOVL C01041 V=800.0 PL=0
MOVL C01042 V=800.0 PL=0
MOVL C01043 V=800.0 PL=0
MOVL C01044 V=800.0 PL=0
MOVL C01045 V=800.0 PL=0
MOVL C01046 V=800.0 PL=0
MOVL C01047 V=800.0 PL=0
MOVL C01048 V=800.0 PL=0
MOVL C01049 V=800.0 PL=0
MOVL C01050 V=800.0 PL=0
MOVL C01051 V=800.0 PL=0
MOVL C01052 V=800.0 PL=0
MOVL C01053 V=800.0 PL=0
MOVL C01054 V=800.0 PL=0
MOVL C01055 V=800.0 PL=0
MOVL C01056 V=800.0 PL=0
MOVL C01057 V=800.0 PL=0
MOVL C01058 V=800.0 PL=0
MOVL C01059 V=800.0 PL=0
MOVL C01060 V=800.0 PL=0
MOVL C01061 V=800.0 PL=0
MOVL C01062 V=800.0 PL=0
MOVL C01063 V=800.0 PL=0
MOVL C01064 V=800.0 PL=0
MOVL C01065 V=800.0 PL=0
MOVL C01066 V=800.0 PL=0
MOVL C01067 V=800.0 PL=0
MOVL C01068 V=800.0 PL=0
MOVL C01069 V=800.0 PL=0
MOVL C01070 V=800.0 PL=0
MOVL C01071 V=800.0 PL=0
MOVL C01072 V=800.0 PL=0
MOVL C01073 V=800.0 PL=0
MOVL C01074 V=800.0 PL=0
MOVL C01075 V=800.0 PL=0
MOVL C01076 V=800.0 PL=0
MOVL C01077 V=800.0 PL=0
MOVL C01078 V=800.0 PL=0
MOVL C01079 V=800.0 PL=0
MOVL C01080 V=800.0 PL=0
MOVL C01081 V=800.0 PL=0
MOVL C01082 V=800.0 PL=0
MOVL C01083 V=800.0 PL=0
MOVL C01084 V=800.0 PL=0
MOVL C01085 V=800.0 PL=0
MOVL C01086 V=800.0 PL=0
MOVL C01087 V=800.0 PL=0
MOVL C01088 V=800.0 PL=0
MOVL C01089 V=800.0 PL=0
MOVL C01090 V=800.0 PL=0
MOVL C01091 V=800.0 PL=0
MOVL C01092 V=800.0 PL=0
MOVL C01093 V=800.0 PL=0
MOVL C01094 V=800.0 PL=0
MOVL C01095 V=800.0 PL=0
MOVL C01096 V=800.0 PL=0
MOVL C01097 V=800.0 PL=0
MOVL C01098 V=800.0 PL=0
MOVL C01099 V=800.0 PL=0
MOVL C01100 V=800.0 PL=0
MOVL C01101 V=800.0 PL=0
MOVL C01102 V=800.0 PL=0
MOVL C01103 V=800.0 PL=0
MOVL C01104 V=800.0 PL=0
MOVL C01105 V=800.0 PL=0
MOVL C01106 V=800.0 PL=0
MOVL C01107 V=800.0 PL=0
MOVL C01108 V=800.0 PL=0
MOVL C01109 V=800.0 PL=0
MOVL C01110 V=800.0 PL=0
MOVL C01111 V=800.0 PL=0
MOVL C01112 V=800.0 PL=0
MOVL C01113 V=800.0 PL=0
MOVL C01114 V=800.0 PL=0
MOVL C01115 V=800.0 PL=0
MOVL C01116 V=800.0 PL=0
MOVL C01117 V=800.0 PL=0
MOVL C01118 V=800.0 PL=0
MOVL C01119 V=800.0 PL=0
MOVL C01120 V=800.0 PL=0
MOVL C01121 V=800.0 PL=0
MOVL C01122 V=800.0 PL=0
MOVL C01123 V=800.0 PL=0
MOVL C01124 V=800.0 PL=0
MOVL C01125 V=800.0 PL=0
MOVL C01126 V=800.0 PL=0
MOVL C01127 V=800.0 PL=0
MOVL C01128 V=800.0 PL=0
MOVL C01129 V=800.0 PL=0
MOVL C01130 V=800.0 PL=0
MOVL C01131 V=800.0 PL=0
MOVL C01132 V=800.0 PL=0
MOVL C01133 V=800.0 PL=0
MOVL C01134 V=800.0 PL=0
MOVL C01135 V=800.0 PL=0
MOVL C01136 V=800.0 PL=0
MOVL C01137 V=800.0 PL=0
MOVL C01138 V=800.0 PL=0
MOVL C01139 V=800.0 PL=0
MOVL C01140 V=800.0 PL=0
MOVL C01141 V=800.0 PL=0
MOVL C01142 V=800.0 PL=0
MOVL C01143 V=800.0 PL=0
MOVL C01144 V=800.0 PL=0
MOVL C01145 V=800.0 PL=0
MOVL C01146 V=800.0 PL=0
MOVL C01147 V=800.0 PL=0
MOVL C01148 V=800.0 PL=0
MOVL C01149 V=800.0 PL=0
MOVL C01150 V=800.0 PL=0
MOVL C01151 V=800.0 PL=0
MOVL C01152 V=800.0 PL=0
MOVL C01153 V=800.0 PL=0
MOVL C01154 V=800.0 PL=0
MOVL C01155 V=800.0 PL=0
MOVL C01156 V=800.0 PL=0
MOVL C01157 V=800.0 PL=0
MOVL C01158 V=800.0 PL=0
MOVL C01159 V=800.0 PL=0
MOVL C01160 V=800.0 PL=0
MOVL C01161 V=800.0 PL=0
MOVL C01162 V=800.0 PL=0
MOVL C01163 V=800.0 PL=0
MOVL C01164 V=800.0 PL=0
MOVL C01165 V=800.0 PL=0
MOVL C01166 V=800.0 PL=0
MOVL C01167 V=800.0 PL=0
MOVL C01168 V=800.0 PL=0
MOVL C01169 V=800.0 PL=0
MOVL C01170 V=800.0 PL=0
MOVL C01171 V=800.0 PL=0
MOVL C01172 V=800.0 PL=0
MOVL C01173 V=800.0 PL=0
MOVL C01174 V=800.0 PL=0
MOVL C01175 V=800.0 PL=0
MOVL C01176 V=800.0 PL=0
MOVL C01177 V=800.0 PL=0
MOVL C01178 V=800.0 PL=0
MOVL C01179 V=800.0 PL=0
MOVL C01180 V=800.0 PL=0
MOVL C01181 V=800.0 PL=0
MOVL C01182 V=800.0 PL=0
MOVL C01183 V=800.0 PL=0
MOVL C01184 V=800.0 PL=0
MOVL C01185 V=800.0 PL=0
MOVL C01186 V=800.0 PL=0
MOVL C01187 V=800.0 PL=0
MOVL C01188 V=800.0 PL=0
MOVL C01189 V=800.0 PL=0
MOVL C01190 V=800.0 PL=0
MOVL C01191 V=800.0 PL=0
MOVL C01192 V=800.0 PL=0
MOVL C01193 V=800.0 PL=0
MOVL C01194 V=800.0 PL=0
MOVL C01195 V=800.0 PL=0
MOVL C01196 V=800.0 PL=0
MOVL C01197 V=800.0 PL=0
MOVL C01198 V=800.0 PL=0
MOVL C01199 V=800.0 PL=0
MOVL C01200 V=800.0 PL=0
MOVL C01201 V=800.0 PL=0
MOVL C01202 V=800.0 PL=0
MOVL C01203 V=800.0 PL=0
MOVL C01204 V=800.0 PL=0
MOVL C01205 V=800.0 PL=0
MOVL C01206 V=800.0 PL=0
MOVL C01207 V=800.0 PL=0
MOVL C01208 V=800.0 PL=0
MOVL C01209 V=800.0 PL=0
MOVL C01210 V=800.0 PL=0
MOVL C01211 V=800.0 PL=0
MOVL C01212 V=800.0 PL=0
MOVL C01213 V=800.0 PL=0
MOVL C01214 V=800.0 PL=0
MOVL C01215 V=800.0 PL=0
MOVL C01216 V=800.0 PL=0
MOVL C01217 V=800.0 PL=0
MOVL C01218 V=800.0 PL=0
MOVL C01219 V=800.0 PL=0
MOVL C01220 V=800.0 PL=0
MOVL C01221 V=800.0 PL=0
MOVL C01222 V=800.0 PL=0
MOVL C01223 V=800.0 PL=0
MOVL C01224 V=800.0 PL=0
MOVL C01225 V=800.0 PL=0
MOVL C01226 V=800.0 PL=0
MOVL C01227 V=800.0 PL=0
MOVL C01228 V=800.0 PL=0
MOVL C01229 V=800.0 PL=0
MOVL C01230 V=800.0 PL=0
MOVL C01231 V=800.0 PL=0
MOVL C01232 V=800.0 PL=0
MOVL C01233 V=800.0 PL=0
MOVL C01234 V=800.0 PL=0
MOVL C01235 V=800.0 PL=0
MOVL C01236 V=800.0 PL=0
MOVL C01237 V=800.0 PL=0
MOVL C01238 V=800.0 PL=0
MOVL C01239 V=800.0 PL=0
MOVL C01240 V=800.0 PL=0
MOVL C01241 V=800.0 PL=0
MOVL C01242 V=800.0 PL=0
MOVL C01243 V=800.0 PL=0
MOVL C01244 V=800.0 PL=0
MOVL C01245 V=800.0 PL=0
MOVL C01246 V=800.0 PL=0
MOVL C01247 V=800.0 PL=0
MOVL C01248 V=800.0 PL=0
MOVL C01249 V=800.0 PL=0
MOVL C01250 V=800.0 PL=0
MOVL C01251 V=800.0 PL=0
MOVL C01252 V=800.0 PL=0
MOVL C01253 V=800.0 PL=0
MOVL C01254 V=800.0 PL=0
MOVL C01255 V=800.0 PL=0
MOVL C01256 V=800.0 PL=0
MOVL C01257 V=800.0 PL=0
MOVL C01258 V=800.0 PL=0
MOVL C01259 V=800.0 PL=0
MOVL C01260 V=800.0 PL=0
MOVL C01261 V=800.0 PL=0
MOVL C01262 V=800.0 PL=0
MOVL C01263 V=800.0 PL=0
MOVL C01264 V=800.0 PL=0
MOVL C01265 V=800.0 PL=0
MOVL C01266 V=800.0 PL=0
MOVL C01267 V=800.0 PL=0
MOVL C01268 V=800.0 PL=0
MOVL C01269 V=800.0 PL=0
MOVL C01270 V=800.0 PL=0
MOVL C01271 V=800.0 PL=0
MOVL C01272 V=800.0 PL=0
MOVL C01273 V=800.0 PL=0
MOVL C01274 V=800.0 PL=0
MOVL C01275 V=800.0 PL=0
MOVL C01276 V=800.0 PL=0
MOVL C01277 V=800.0 PL=0
MOVL C01278 V=800.0 PL=0
MOVL C01279 V=800.0 PL=0
MOVL C01280 V=800.0 PL=0
MOVL C01281 V=800.0 PL=0
MOVL C01282 V=800.0 PL=0
MOVL C01283 V=800.0 PL=0
MOVL C01284 V=800.0 PL=0
MOVL C01285 V=800.0 PL=0
MOVL C01286 V=800.0 PL=0
MOVL C01287 V=800.0 PL=0
MOVL C01288 V=800.0 PL=0
MOVL C01289 V=800.0 PL=0
MOVL C01290 V=800.0 PL=0
MOVL C01291 V=800.0 PL=0
MOVL C01292 V=800.0 PL=0
MOVL C01293 V=800.0 PL=0
MOVL C01294 V=800.0 PL=0
MOVL C01295 V=800.0 PL=0
MOVL C01296 V=800.0 PL=0
MOVL C01297 V=800.0 PL=0
MOVL C01298 V=800.0 PL=0
MOVL C01299 V=800.0 PL=0
MOVL C01300 V=800.0 PL=0
MOVL C01301 V=800.0 PL=0
MOVL C01302 V=800.0 PL=0
MOVL C01303 V=800.0 PL=0
MOVL C01304 V=800.0 PL=0
MOVL C01305 V=800.0 PL=0
MOVL C01306 V=800.0 PL=0
MOVL C01307 V=800.0 PL=0
MOVL C01308 V=800.0 PL=0
MOVL C01309 V=800.0 PL=0
MOVL C01310 V=800.0 PL=0
MOVL C01311 V=800.0 PL=0
MOVL C01312 V=800.0 PL=0
MOVL C01313 V=800.0 PL=0
MOVL C01314 V=800.0 PL=0
MOVL C01315 V=800.0 PL=0
MOVL C01316 V=800.0 PL=0
MOVL C01317 V=800.0 PL=0
MOVL C01318 V=800.0 PL=0
MOVL C01319 V=800.0 PL=0
MOVL C01320 V=800.0 PL=0
MOVL C01321 V=800.0 PL=0
MOVL C01322 V=800.0 PL=0
MOVL C01323 V=800.0 PL=0
MOVL C01324 V=800.0 PL=0
MOVL C01325 V=800.0 PL=0
MOVL C01326 V=800.0 PL=0
MOVL C01327 V=800.0 PL=0
MOVL C01328 V=800.0 PL=0
MOVL C01329 V=800.0 PL=0
MOVL C01330 V=800.0 PL=0
MOVL C01331 V=800.0 PL=0
MOVL C01332 V=800.0 PL=0
MOVL C01333 V=800.0 PL=0
MOVL C01334 V=800.0 PL=0
MOVL C01335 V=800.0 PL=0
MOVL C01336 V=800.0 PL=0
MOVL C01337 V=800.0 PL=0
MOVL C01338 V=800.0 PL=0
MOVL C01339 V=800.0 PL=0
MOVL C01340 V=800.0 PL=0
MOVL C01341 V=800.0 PL=0
MOVL C01342 V=800.0 PL=0
MOVL C01343 V=800.0 PL=0
MOVL C01344 V=800.0 PL=0
MOVL C01345 V=800.0 PL=0
MOVL C01346 V=800.0 PL=0
MOVL C01347 V=800.0 PL=0
MOVL C01348 V=800.0 PL=0
MOVL C01349 V=800.0 PL=0
MOVL C01350 V=800.0 PL=0
MOVL C01351 V=800.0 PL=0
MOVL C01352 V=800.0 PL=0
MOVL C01353 V=800.0 PL=0
MOVL C01354 V=800.0 PL=0
MOVL C01355 V=800.0 PL=0
MOVL C01356 V=800.0 PL=0
MOVL C01357 V=800.0 PL=0
MOVL C01358 V=800.0 PL=0
MOVL C01359 V=800.0 PL=0
MOVL C01360 V=800.0 PL=0
MOVL C01361 V=800.0 PL=0
MOVL C01362 V=800.0 PL=0
MOVL C01363 V=800.0 PL=0
MOVL C01364 V=800.0 PL=0
MOVL C01365 V=800.0 PL=0
MOVL C01366 V=800.0 PL=0
MOVL C01367 V=800.0 PL=0
MOVL C01368 V=800.0 PL=0
MOVL C01369 V=800.0 PL=0
MOVL C01370 V=800.0 PL=0
MOVL C01371 V=800.0 PL=0
MOVL C01372 V=800.0 PL=0
MOVL C01373 V=800.0 PL=0
MOVL C01374 V=800.0 PL=0
MOVL C01375 V=800.0 PL=0
MOVL C01376 V=800.0 PL=0
MOVL C01377 V=800.0 PL=0
MOVL C01378 V=800.0 PL=0
MOVL C01379 V=800.0 PL=0
MOVL C01380 V=800.0 PL=0
MOVL C01381 V=800.0 PL=0
MOVL C01382 V=800.0 PL=0
MOVL C01383 V=800.0 PL=0
MOVL C01384 V=800.0 PL=0
MOVL C01385 V=800.0 PL=0
MOVL C01386 V=800.0 PL=0
MOVL C01387 V=800.0 PL=0
MOVL C01388 V=800.0 PL=0
MOVL C01389 V=800.0 PL=0
MOVL C01390 V=800.0 PL=0
MOVL C01391 V=800.0 PL=0
MOVL C01392 V=800.0 PL=0
MOVL C01393 V=800.0 PL=0
MOVL C01394 V=800.0 PL=0
MOVL C01395 V=800.0 PL=0
MOVL C01396 V=800.0 PL=0
MOVL C01397 V=800.0 PL=0
MOVL C01398 V=800.0 PL=0
MOVL C01399 V=800.0 PL=0
MOVL C01400 V=800.0 PL=0
MOVL C01401 V=800.0 PL=0
MOVL C01402 V=800.0 PL=0
MOVL C01403 V=800.0 PL=0
MOVL C01404 V=800.0 PL=0
MOVL C01405 V=800.0 PL=0
MOVL C01406 V=800.0 PL=0
MOVL C01407 V=800.0 PL=0
MOVL C01408 V=800.0 PL=0
MOVL C01409 V=800.0 PL=0
MOVL C01410 V=800.0 PL=0
MOVL C01411 V=800.0 PL=0
MOVL C01412 V=800.0 PL=0
MOVL C01413 V=800.0 PL=0
MOVL C01414 V=800.0 PL=0
MOVL C01415 V=800.0 PL=0
MOVL C01416 V=800.0 PL=0
MOVL C01417 V=800.0 PL=0
MOVL C01418 V=800.0 PL=0
MOVL C01419 V=800.0 PL=0
MOVL C01420 V=800.0 PL=0
MOVL C01421 V=800.0 PL=0
MOVL C01422 V=800.0 PL=0
MOVL C01423 V=800.0 PL=0
MOVL C01424 V=800.0 PL=0
MOVL C01425 V=800.0 PL=0
MOVL C01426 V=800.0 PL=0
MOVL C01427 V=800.0 PL=0
MOVL C01428 V=800.0 PL=0
MOVL C01429 V=800.0 PL=0
MOVL C01430 V=800.0 PL=0
MOVL C01431 V=800.0 PL=0
MOVL C01432 V=800.0 PL=0
MOVL C01433 V=800.0 PL=0
MOVL C01434 V=800.0 PL=0
MOVL C01435 V=800.0 PL=0
MOVL C01436 V=800.0 PL=0
MOVL C01437 V=800.0 PL=0
MOVL C01438 V=800.0 PL=0
MOVL C01439 V=800.0 PL=0
MOVL C01440 V=800.0 PL=0
MOVL C01441 V=800.0 PL=0
MOVL C01442 V=800.0 PL=0
MOVL C01443 V=800.0 PL=0
MOVL C01444 V=800.0 PL=0
MOVL C01445 V=800.0 PL=0
MOVL C01446 V=800.0 PL=0
MOVL C01447 V=800.0 PL=0
MOVL C01448 V=800.0 PL=0
MOVL C01449 V=800.0 PL=0
MOVL C01450 V=800.0 PL=0
MOVL C01451 V=800.0 PL=0
MOVL C01452 V=800.0 PL=0
MOVL C01453 V=800.0 PL=0
MOVL C01454 V=800.0 PL=0
MOVL C01455 V=800.0 PL=0
MOVL C01456 V=800.0 PL=0
MOVL C01457 V=800.0 PL=0
MOVL C01458 V=800.0 PL=0
MOVL C01459 V=800.0 PL=0
MOVL C01460 V=800.0 PL=0
MOVL C01461 V=800.0 PL=0
MOVL C01462 V=800.0 PL=0
MOVL C01463 V=800.0 PL=0
MOVL C01464 V=800.0 PL=0
MOVL C01465 V=800.0 PL=0
MOVL C01466 V=800.0 PL=0
MOVL C01467 V=800.0 PL=0
MOVL C01468 V=800.0 PL=0
MOVL C01469 V=800.0 PL=0
MOVL C01470 V=800.0 PL=0
MOVL C01471 V=800.0 PL=0
MOVL C01472 V=800.0 PL=0
MOVL C01473 V=800.0 PL=0
MOVL C01474 V=800.0 PL=0
MOVL C01475 V=800.0 PL=0
MOVL C01476 V=800.0 PL=0
MOVL C01477 V=800.0 PL=0
MOVL C01478 V=800.0 PL=0
MOVL C01479 V=800.0 PL=0
MOVL C01480 V=800.0 PL=0
MOVL C01481 V=800.0 PL=0
MOVL C01482 V=800.0 PL=0
MOVL C01483 V=800.0 PL=0
MOVL C01484 V=800.0 PL=0
MOVL C01485 V=800.0 PL=0
MOVL C01486 V=800.0 PL=0
MOVL C01487 V=800.0 PL=0
MOVL C01488 V=800.0 PL=0
MOVL C01489 V=800.0 PL=0
MOVL C01490 V=800.0 PL=0
MOVL C01491 V=800.0 PL=0
MOVL C01492 V=800.0 PL=0
MOVL C01493 V=800.0 PL=0
MOVL C01494 V=800.0 PL=0
MOVL C01495 V=800.0 PL=0
MOVL C01496 V=800.0 PL=0
MOVL C01497 V=800.0 PL=0
MOVL C01498 V=800.0 PL=0
MOVL C01499 V=800.0 PL=0
MOVL C01500 V=800.0 PL=0
MOVL C01501 V=800.0 PL=0
MOVL C01502 V=800.0 PL=0
MOVL C01503 V=800.0 PL=0
MOVL C01504 V=800.0 PL=0
MOVL C01505 V=800.0 PL=0
MOVL C01506 V=800.0 PL=0
MOVL C01507 V=800.0 PL=0
MOVL C01508 V=800.0 PL=0
MOVL C01509 V=800.0 PL=0
MOVL C01510 V=800.0 PL=0
MOVL C01511 V=800.0 PL=0
MOVL C01512 V=800.0 PL=0
MOVL C01513 V=800.0 PL=0
MOVL C01514 V=800.0 PL=0
MOVL C01515 V=800.0 PL=0
MOVL C01516 V=800.0 PL=0
MOVL C01517 V=800.0 PL=0
MOVL C01518 V=800.0 PL=0
MOVL C01519 V=800.0 PL=0
MOVL C01520 V=800.0 PL=0
MOVL C01521 V=800.0 PL=0
MOVL C01522 V=800.0 PL=0
MOVL C01523 V=800.0 PL=0
MOVL C01524 V=800.0 PL=0
MOVL C01525 V=800.0 PL=0
MOVL C01526 V=800.0 PL=0
MOVL C01527 V=800.0 PL=0
MOVL C01528 V=800.0 PL=0
MOVL C01529 V=800.0 PL=0
MOVL C01530 V=800.0 PL=0
MOVL C01531 V=800.0 PL=0
MOVL C01532 V=800.0 PL=0
MOVL C01533 V=800.0 PL=0
MOVL C01534 V=800.0 PL=0
MOVL C01535 V=800.0 PL=0
MOVL C01536 V=800.0 PL=0
MOVL C01537 V=800.0 PL=0
MOVL C01538 V=800.0 PL=0
MOVL C01539 V=800.0 PL=0
MOVL C01540 V=800.0 PL=0
MOVL C01541 V=800.0 PL=0
MOVL C01542 V=800.0 PL=0
MOVL C01543 V=800.0 PL=0
MOVL C01544 V=800.0 PL=0
MOVL C01545 V=800.0 PL=0
MOVL C01546 V=800.0 PL=0
MOVL C01547 V=800.0 PL=0
MOVL C01548 V=800.0 PL=0
MOVL C01549 V=800.0 PL=0
MOVL C01550 V=800.0 PL=0
MOVL C01551 V=800.0 PL=0
MOVL C01552 V=800.0 PL=0
MOVL C01553 V=800.0 PL=0
MOVL C01554 V=800.0 PL=0
MOVL C01555 V=800.0 PL=0
MOVL C01556 V=800.0 PL=0
MOVL C01557 V=800.0 PL=0
MOVL C01558 V=800.0 PL=0
MOVL C01559 V=800.0 PL=0
MOVL C01560 V=800.0 PL=0
MOVL C01561 V=800.0 PL=0
MOVL C01562 V=800.0 PL=0
MOVL C01563 V=800.0 PL=0
MOVL C01564 V=800.0 PL=0
MOVL C01565 V=800.0 PL=0
MOVL C01566 V=800.0 PL=0
MOVL C01567 V=800.0 PL=0
MOVL C01568 V=800.0 PL=0
MOVL C01569 V=800.0 PL=0
MOVL C01570 V=800.0 PL=0
MOVL C01571 V=800.0 PL=0
MOVL C01572 V=800.0 PL=0
MOVL C01573 V=800.0 PL=0
MOVL C01574 V=800.0 PL=0
MOVL C01575 V=800.0 PL=0
MOVL C01576 V=800.0 PL=0
MOVL C01577 V=800.0 PL=0
MOVL C01578 V=800.0 PL=0
MOVL C01579 V=800.0 PL=0
MOVL C01580 V=800.0 PL=0
MOVL C01581 V=800.0 PL=0
MOVL C01582 V=800.0 PL=0
MOVL C01583 V=800.0 PL=0
MOVL C01584 V=800.0 PL=0
MOVL C01585 V=800.0 PL=0
MOVL C01586 V=800.0 PL=0
MOVL C01587 V=800.0 PL=0
MOVL C01588 V=800.0 PL=0
MOVL C01589 V=800.0 PL=0
MOVL C01590 V=800.0 PL=0
MOVL C01591 V=800.0 PL=0
MOVL C01592 V=800.0 PL=0
MOVL C01593 V=800.0 PL=0
MOVL C01594 V=800.0 PL=0
MOVL C01595 V=800.0 PL=0
MOVL C01596 V=800.0 PL=0
MOVL C01597 V=800.0 PL=0
MOVL C01598 V=800.0 PL=0
MOVL C01599 V=800.0 PL=0
MOVL C01600 V=800.0 PL=0
MOVL C01601 V=800.0 PL=0
MOVL C01602 V=800.0 PL=0
MOVL C01603 V=800.0 PL=0
MOVL C01604 V=800.0 PL=0
MOVL C01605 V=800.0 PL=0
MOVL C01606 V=800.0 PL=0
MOVL C01607 V=800.0 PL=0
MOVL C01608 V=800.0 PL=0
MOVL C01609 V=800.0 PL=0
MOVL C01610 V=800.0 PL=0
MOVL C01611 V=800.0 PL=0
MOVL C01612 V=800.0 PL=0
MOVL C01613 V=800.0 PL=0
MOVL C01614 V=800.0 PL=0
MOVL C01615 V=800.0 PL=0
MOVL C01616 V=800.0 PL=0
MOVL C01617 V=800.0 PL=0
MOVL C01618 V=800.0 PL=0
MOVL C01619 V=800.0 PL=0
MOVL C01620 V=800.0 PL=0
MOVL C01621 V=800.0 PL=0
MOVL C01622 V=800.0 PL=0
MOVL C01623 V=800.0 PL=0
MOVL C01624 V=800.0 PL=0
MOVL C01625 V=800.0 PL=0
MOVL C01626 V=800.0 PL=0
MOVL C01627 V=800.0 PL=0
MOVL C01628 V=800.0 PL=0
MOVL C01629 V=800.0 PL=0
MOVL C01630 V=800.0 PL=0
MOVL C01631 V=800.0 PL=0
MOVL C01632 V=800.0 PL=0
MOVL C01633 V=800.0 PL=0
MOVL C01634 V=800.0 PL=0
MOVL C01635 V=800.0 PL=0
MOVL C01636 V=800.0 PL=0
MOVL C01637 V=800.0 PL=0
MOVL C01638 V=800.0 PL=0
MOVL C01639 V=800.0 PL=0
MOVL C01640 V=800.0 PL=0
MOVL C01641 V=800.0 PL=0
MOVL C01642 V=800.0 PL=0
MOVL C01643 V=800.0 PL=0
MOVL C01644 V=800.0 PL=0
MOVL C01645 V=800.0 PL=0
MOVL C01646 V=800.0 PL=0
MOVL C01647 V=800.0 PL=0
MOVL C01648 V=800.0 PL=0
MOVL C01649 V=800.0 PL=0
MOVL C01650 V=800.0 PL=0
MOVL C01651 V=800.0 PL=0
MOVL C01652 V=800.0 PL=0
MOVL C01653 V=800.0 PL=0
MOVL C01654 V=800.0 PL=0
MOVL C01655 V=800.0 PL=0
MOVL C01656 V=800.0 PL=0
MOVL C01657 V=800.0 PL=0
MOVL C01658 V=800.0 PL=0
MOVL C01659 V=800.0 PL=0
MOVL C01660 V=800.0 PL=0
MOVL C01661 V=800.0 PL=0
MOVL C01662 V=800.0 PL=0
MOVL C01663 V=800.0 PL=0
MOVL C01664 V=800.0 PL=0
MOVL C01665 V=800.0 PL=0
MOVL C01666 V=800.0 PL=0
MOVL C01667 V=800.0 PL=0
MOVL C01668 V=800.0 PL=0
MOVL C01669 V=800.0 PL=0
MOVL C01670 V=800.0 PL=0
MOVL C01671 V=800.0 PL=0
MOVL C01672 V=800.0 PL=0
MOVL C01673 V=800.0 PL=0
MOVL C01674 V=800.0 PL=0
MOVL C01675 V=800.0 PL=0
MOVL C01676 V=800.0 PL=0
MOVL C01677 V=800.0 PL=0
MOVL C01678 V=800.0 PL=0
MOVL C01679 V=800.0 PL=0
MOVL C01680 V=800.0 PL=0
MOVL C01681 V=800.0 PL=0
MOVL C01682 V=800.0 PL=0
MOVL C01683 V=800.0 PL=0
MOVL C01684 V=800.0 PL=0
MOVL C01685 V=800.0 PL=0
MOVL C01686 V=800.0 PL=0
MOVL C01687 V=800.0 PL=0
MOVL C01688 V=800.0 PL=0
MOVL C01689 V=800.0 PL=0
MOVL C01690 V=800.0 PL=0
MOVL C01691 V=800.0 PL=0
MOVL C01692 V=800.0 PL=0
MOVL C01693 V=800.0 PL=0
MOVL C01694 V=800.0 PL=0
MOVL C01695 V=800.0 PL=0
MOVL C01696 V=800.0 PL=0
MOVL C01697 V=800.0 PL=0
MOVL C01698 V=800.0 PL=0
MOVL C01699 V=800.0 PL=0
MOVL C01700 V=800.0 PL=0
MOVL C01701 V=800.0 PL=0
MOVL C01702 V=800.0 PL=0
MOVL C01703 V=800.0 PL=0
MOVL C01704 V=800.0 PL=0
MOVL C01705 V=800.0 PL=0
MOVL C01706 V=800.0 PL=0
MOVL C01707 V=800.0 PL=0
MOVL C01708 V=800.0 PL=0
MOVL C01709 V=800.0 PL=0
MOVL C01710 V=800.0 PL=0
MOVL C01711 V=800.0 PL=0
MOVL C01712 V=800.0 PL=0
MOVL C01713 V=800.0 PL=0
MOVL C01714 V=800.0 PL=0
MOVL C01715 V=800.0 PL=0
MOVL C01716 V=800.0 PL=0
MOVL C01717 V=800.0 PL=0
MOVL C01718 V=800.0 PL=0
MOVL C01719 V=800.0 PL=0
MOVL C01720 V=800.0 PL=0
MOVL C01721 V=800.0 PL=0
MOVL C01722 V=800.0 PL=0
MOVL C01723 V=800.0 PL=0
MOVL C01724 V=800.0 PL=0
MOVL C01725 V=800.0 PL=0
MOVL C01726 V=800.0 PL=0
MOVL C01727 V=800.0 PL=0
MOVL C01728 V=800.0 PL=0
MOVL C01729 V=800.0 PL=0
MOVL C01730 V=800.0 PL=0
MOVL C01731 V=800.0 PL=0
MOVL C01732 V=800.0 PL=0
MOVL C01733 V=800.0 PL=0
MOVL C01734 V=800.0 PL=0
MOVL C01735 V=800.0 PL=0
MOVL C01736 V=800.0 PL=0
MOVL C01737 V=800.0 PL=0
MOVL C01738 V=800.0 PL=0
MOVL C01739 V=800.0 PL=0
MOVL C01740 V=800.0 PL=0
MOVL C01741 V=800.0 PL=0
MOVL C01742 V=800.0 PL=0
MOVL C01743 V=800.0 PL=0
MOVL C01744 V=800.0 PL=0
MOVL C01745 V=800.0 PL=0
MOVL C01746 V=800.0 PL=0
MOVL C01747 V=800.0 PL=0
MOVL C01748 V=800.0 PL=0
MOVL C01749 V=800.0 PL=0
MOVL C01750 V=800.0 PL=0
MOVL C01751 V=800.0 PL=0
MOVL C01752 V=800.0 PL=0
MOVL C01753 V=800.0 PL=0
MOVL C01754 V=800.0 PL=0
MOVL C01755 V=800.0 PL=0
MOVL C01756 V=800.0 PL=0
MOVL C01757 V=800.0 PL=0
MOVL C01758 V=800.0 PL=0
MOVL C01759 V=800.0 PL=0
MOVL C01760 V=800.0 PL=0
MOVL C01761 V=800.0 PL=0
MOVL C01762 V=800.0 PL=0
MOVL C01763 V=800.0 PL=0
MOVL C01764 V=800.0 PL=0
MOVL C01765 V=800.0 PL=0
MOVL C01766 V=800.0 PL=0
MOVL C01767 V=800.0 PL=0
MOVL C01768 V=800.0 PL=0
MOVL C01769 V=800.0 PL=0
MOVL C01770 V=800.0 PL=0
MOVL C01771 V=800.0 PL=0
MOVL C01772 V=800.0 PL=0
MOVL C01773 V=800.0 PL=0
MOVL C01774 V=800.0 PL=0
MOVL C01775 V=800.0 PL=0
MOVL C01776 V=800.0 PL=0
MOVL C01777 V=800.0 PL=0
MOVL C01778 V=800.0 PL=0
MOVL C01779 V=800.0 PL=0
MOVL C01780 V=800.0 PL=0
MOVL C01781 V=800.0 PL=0
MOVL C01782 V=800.0 PL=0
MOVL C01783 V=800.0 PL=0
MOVL C01784 V=800.0 PL=0
MOVL C01785 V=800.0 PL=0
MOVL C01786 V=800.0 PL=0
MOVL C01787 V=800.0 PL=0
MOVL C01788 V=800.0 PL=0
MOVL C01789 V=800.0 PL=0
MOVL C01790 V=800.0 PL=0
MOVL C01791 V=800.0 PL=0
MOVL C01792 V=800.0 PL=0
MOVL C01793 V=800.0 PL=0
MOVL C01794 V=800.0 PL=0
MOVL C01795 V=800.0 PL=0
MOVL C01796 V=800.0 PL=0
MOVL C01797 V=800.0 PL=0
MOVL C01798 V=800.0 PL=0
MOVL C01799 V=800.0 PL=0
MOVL C01800 V=800.0 PL=0
MOVL C01801 V=800.0 PL=0
MOVL C01802 V=800.0 PL=0
MOVL C01803 V=800.0 PL=0
MOVL C01804 V=800.0 PL=0
MOVL C01805 V=800.0 PL=0
MOVL C01806 V=800.0 PL=0
MOVL C01807 V=800.0 PL=0
MOVL C01808 V=800.0 PL=0
MOVL C01809 V=800.0 PL=0
MOVL C01810 V=800.0 PL=0
MOVL C01811 V=800.0 PL=0
MOVL C01812 V=800.0 PL=0
MOVL C01813 V=800.0 PL=0
MOVL C01814 V=800.0 PL=0
MOVL C01815 V=800.0 PL=0
MOVL C01816 V=800.0 PL=0
MOVL C01817 V=800.0 PL=0
MOVL C01818 V=800.0 PL=0
MOVL C01819 V=800.0 PL=0
MOVL C01820 V=800.0 PL=0
MOVL C01821 V=800.0 PL=0
MOVL C01822 V=800.0 PL=0
MOVL C01823 V=800.0 PL=0
MOVL C01824 V=800.0 PL=0
MOVL C01825 V=800.0 PL=0
MOVL C01826 V=800.0 PL=0
MOVL C01827 V=800.0 PL=0
MOVL C01828 V=800.0 PL=0
MOVL C01829 V=800.0 PL=0
MOVL C01830 V=800.0 PL=0
MOVL C01831 V=800.0 PL=0
MOVL C01832 V=800.0 PL=0
MOVL C01833 V=800.0 PL=0
MOVL C01834 V=800.0 PL=0
MOVL C01835 V=800.0 PL=0
MOVL C01836 V=800.0 PL=0
MOVL C01837 V=800.0 PL=0
MOVL C01838 V=800.0 PL=0
MOVL C01839 V=800.0 PL=0
MOVL C01840 V=800.0 PL=0
MOVL C01841 V=800.0 PL=0
MOVL C01842 V=800.0 PL=0
MOVL C01843 V=800.0 PL=0
MOVL C01844 V=800.0 PL=0
MOVL C01845 V=800.0 PL=0
MOVL C01846 V=800.0 PL=0
MOVL C01847 V=800.0 PL=0
MOVL C01848 V=800.0 PL=0
MOVL C01849 V=800.0 PL=0
MOVL C01850 V=800.0 PL=0
MOVL C01851 V=800.0 PL=0
MOVL C01852 V=800.0 PL=0
MOVL C01853 V=800.0 PL=0
MOVL C01854 V=800.0 PL=0
MOVL C01855 V=800.0 PL=0
MOVL C01856 V=800.0 PL=0
MOVL C01857 V=800.0 PL=0
MOVL C01858 V=800.0 PL=0
MOVL C01859 V=800.0 PL=0
MOVL C01860 V=800.0 PL=0
MOVL C01861 V=800.0 PL=0
MOVL C01862 V=800.0 PL=0
MOVL C01863 V=800.0 PL=0
MOVL C01864 V=800.0 PL=0
MOVL C01865 V=800.0 PL=0
MOVL C01866 V=800.0 PL=0
MOVL C01867 V=800.0 PL=0
MOVL C01868 V=800.0 PL=0
MOVL C01869 V=800.0 PL=0
MOVL C01870 V=800.0 PL=0
MOVL C01871 V=800.0 PL=0
MOVL C01872 V=800.0 PL=0
MOVL C01873 V=800.0 PL=0
MOVL C01874 V=800.0 PL=0
MOVL C01875 V=800.0 PL=0
MOVL C01876 V=800.0 PL=0
MOVL C01877 V=800.0 PL=0
MOVL C01878 V=800.0 PL=0
MOVL C01879 V=800.0 PL=0
MOVL C01880 V=800.0 PL=0
MOVL C01881 V=800.0 PL=0
MOVL C01882 V=800.0 PL=0
MOVL C01883 V=800.0 PL=0
MOVL C01884 V=800.0 PL=0
MOVL C01885 V=800.0 PL=0
MOVL C01886 V=800.0 PL=0
MOVL C01887 V=800.0 PL=0
MOVL C01888 V=800.0 PL=0
MOVL C01889 V=800.0 PL=0
MOVL C01890 V=800.0 PL=0
MOVL C01891 V=800.0 PL=0
MOVL C01892 V=800.0 PL=0
MOVL C01893 V=800.0 PL=0
MOVL C01894 V=800.0 PL=0
MOVL C01895 V=800.0 PL=0
MOVL C01896 V=800.0 PL=0
MOVL C01897 V=800.0 PL=0
MOVL C01898 V=800.0 PL=0
MOVL C01899 V=800.0 PL=0
MOVL C01900 V=800.0 PL=0
MOVL C01901 V=800.0 PL=0
MOVL C01902 V=800.0 PL=0
MOVL C01903 V=800.0 PL=0
MOVL C01904 V=800.0 PL=0
MOVL C01905 V=800.0 PL=0
MOVL C01906 V=800.0 PL=0
MOVL C01907 V=800.0 PL=0
MOVL C01908 V=800.0 PL=0
MOVL C01909 V=800.0 PL=0
MOVL C01910 V=800.0 PL=0
MOVL C01911 V=800.0 PL=0
MOVL C01912 V=800.0 PL=0
MOVL C01913 V=800.0 PL=0
MOVL C01914 V=800.0 PL=0
MOVL C01915 V=800.0 PL=0
MOVL C01916 V=800.0 PL=0
MOVL C01917 V=800.0 PL=0
MOVL C01918 V=800.0 PL=0
MOVL C01919 V=800.0 PL=0
MOVL C01920 V=800.0 PL=0
MOVL C01921 V=800.0 PL=0
MOVL C01922 V=800.0 PL=0
MOVL C01923 V=800.0 PL=0
MOVL C01924 V=800.0 PL=0
MOVL C01925 V=800.0 PL=0
MOVL C01926 V=800.0 PL=0
MOVL C01927 V=800.0 PL=0
MOVL C01928 V=800.0 PL=0
MOVL C01929 V=800.0 PL=0
MOVL C01930 V=800.0 PL=0
MOVL C01931 V=800.0 PL=0
MOVL C01932 V=800.0 PL=0
MOVL C01933 V=800.0 PL=0
MOVL C01934 V=800.0 PL=0
MOVL C01935 V=800.0 PL=0
MOVL C01936 V=800.0 PL=0
MOVL C01937 V=800.0 PL=0
MOVL C01938 V=800.0 PL=0
MOVL C01939 V=800.0 PL=0
MOVL C01940 V=800.0 PL=0
MOVL C01941 V=800.0 PL=0
MOVL C01942 V=800.0 PL=0
MOVL C01943 V=800.0 PL=0
MOVL C01944 V=800.0 PL=0
MOVL C01945 V=800.0 PL=0
MOVL C01946 V=800.0 PL=0
MOVL C01947 V=800.0 PL=0
MOVL C01948 V=800.0 PL=0
MOVL C01949 V=800.0 PL=0
MOVL C01950 V=800.0 PL=0
MOVL C01951 V=800.0 PL=0
MOVL C01952 V=800.0 PL=0
MOVL C01953 V=800.0 PL=0
MOVL C01954 V=800.0 PL=0
MOVL C01955 V=800.0 PL=0
MOVL C01956 V=800.0 PL=0
MOVL C01957 V=800.0 PL=0
MOVL C01958 V=800.0 PL=0
MOVL C01959 V=800.0 PL=0
MOVL C01960 V=800.0 PL=0
MOVL C01961 V=800.0 PL=0
MOVL C01962 V=800.0 PL=0
MOVL C01963 V=800.0 PL=0
MOVL C01964 V=800.0 PL=0
MOVL C01965 V=800.0 PL=0
MOVL C01966 V=800.0 PL=0
MOVL C01967 V=800.0 PL=0
MOVL C01968 V=800.0 PL=0
MOVL C01969 V=800.0 PL=0
MOVL C01970 V=800.0 PL=0
MOVL C01971 V=800.0 PL=0
MOVL C01972 V=800.0 PL=0
MOVL C01973 V=800.0 PL=0
MOVL C01974 V=800.0 PL=0
MOVL C01975 V=800.0 PL=0
MOVL C01976 V=800.0 PL=0
MOVL C01977 V=800.0 PL=0
MOVL C01978 V=800.0 PL=0
MOVL C01979 V=800.0 PL=0
MOVL C01980 V=800.0 PL=0
MOVL C01981 V=800.0 PL=0
MOVL C01982 V=800.0 PL=0
MOVL C01983 V=800.0 PL=0
MOVL C01984 V=800.0 PL=0
MOVL C01985 V=800.0 PL=0
MOVL C01986 V=800.0 PL=0
MOVL C01987 V=800.0 PL=0
MOVL C01988 V=800.0 PL=0
MOVL C01989 V=800.0 PL=0
MOVL C01990 V=800.0 PL=0
MOVL C01991 V=800.0 PL=0
MOVL C01992 V=800.0 PL=0
MOVL C01993 V=800.0 PL=0
MOVL C01994 V=800.0 PL=0
MOVL C01995 V=800.0 PL=0
MOVL C01996 V=800.0 PL=0
MOVL C01997 V=800.0 PL=0
MOVL C01998 V=800.0 PL=0
MOVL C01999 V=800.0 PL=0
MOVL C02000 V=800.0 PL=0
MOVL C02001 V=800.0 PL=0
MOVL C02002 V=800.0 PL=0
MOVL C02003 V=800.0 PL=0
MOVL C02004 V=800.0 PL=0
MOVL C02005 V=800.0 PL=0
MOVL C02006 V=800.0 PL=0
MOVL C02007 V=800.0 PL=0
MOVL C02008 V=800.0 PL=0
MOVL C02009 V=800.0 PL=0
MOVL C02010 V=800.0 PL=0
MOVL C02011 V=800.0 PL=0
MOVL C02012 V=800.0 PL=0
MOVL C02013 V=800.0 PL=0
MOVL C02014 V=800.0 PL=0
MOVL C02015 V=800.0 PL=0
MOVL C02016 V=800.0 PL=0
MOVL C02017 V=800.0 PL=0
MOVL C02018 V=800.0 PL=0
MOVL C02019 V=800.0 PL=0
MOVL C02020 V=800.0 PL=0
MOVL C02021 V=800.0 PL=0
MOVL C02022 V=800.0 PL=0
MOVL C02023 V=800.0 PL=0
MOVL C02024 V=800.0 PL=0
MOVL C02025 V=800.0 PL=0
MOVL C02026 V=800.0 PL=0
MOVL C02027 V=800.0 PL=0
MOVL C02028 V=800.0 PL=0
MOVL C02029 V=800.0 PL=0
MOVL C02030 V=800.0 PL=0
MOVL C02031 V=800.0 PL=0
MOVL C02032 V=800.0 PL=0
MOVL C02033 V=800.0 PL=0
MOVL C02034 V=800.0 PL=0
MOVL C02035 V=800.0 PL=0
MOVL C02036 V=800.0 PL=0
MOVL C02037 V=800.0 PL=0
MOVL C02038 V=800.0 PL=0
MOVL C02039 V=800.0 PL=0
MOVL C02040 V=800.0 PL=0
MOVL C02041 V=800.0 PL=0
MOVL C02042 V=800.0 PL=0
MOVL C02043 V=800.0 PL=0
MOVL C02044 V=800.0 PL=0
MOVL C02045 V=800.0 PL=0
MOVL C02046 V=800.0 PL=0
MOVL C02047 V=800.0 PL=0
MOVL C02048 V=800.0 PL=0
MOVL C02049 V=800.0 PL=0
MOVL C02050 V=800.0 PL=0
MOVL C02051 V=800.0 PL=0
MOVL C02052 V=800.0 PL=0
MOVL C02053 V=800.0 PL=0
MOVL C02054 V=800.0 PL=0
MOVL C02055 V=800.0 PL=0
MOVL C02056 V=800.0 PL=0
MOVL C02057 V=800.0 PL=0
MOVL C02058 V=800.0 PL=0
MOVL C02059 V=800.0 PL=0
MOVL C02060 V=800.0 PL=0
MOVL C02061 V=800.0 PL=0
MOVL C02062 V=800.0 PL=0
MOVL C02063 V=800.0 PL=0
MOVL C02064 V=800.0 PL=0
MOVL C02065 V=800.0 PL=0
MOVL C02066 V=800.0 PL=0
MOVL C02067 V=800.0 PL=0
MOVL C02068 V=800.0 PL=0
MOVL C02069 V=800.0 PL=0
MOVL C02070 V=800.0 PL=0
MOVL C02071 V=800.0 PL=0
MOVL C02072 V=800.0 PL=0
MOVL C02073 V=800.0 PL=0
MOVL C02074 V=800.0 PL=0
MOVL C02075 V=800.0 PL=0
MOVL C02076 V=800.0 PL=0
MOVL C02077 V=800.0 PL=0
MOVL C02078 V=800.0 PL=0
MOVL C02079 V=800.0 PL=0
MOVL C02080 V=800.0 PL=0
MOVL C02081 V=800.0 PL=0
MOVL C02082 V=800.0 PL=0
MOVL C02083 V=800.0 PL=0
MOVL C02084 V=800.0 PL=0
MOVL C02085 V=800.0 PL=0
MOVL C02086 V=800.0 PL=0
MOVL C02087 V=800.0 PL=0
MOVL C02088 V=800.0 PL=0
MOVL C02089 V=800.0 PL=0
MOVL C02090 V=800.0 PL=0
MOVL C02091 V=800.0 PL=0
MOVL C02092 V=800.0 PL=0
MOVL C02093 V=800.0 PL=0
MOVL C02094 V=800.0 PL=0
MOVL C02095 V=800.0 PL=0
MOVL C02096 V=800.0 PL=0
MOVL C02097 V=800.0 PL=0
MOVL C02098 V=800.0 PL=0
MOVL C02099 V=800.0 PL=0
MOVL C02100 V=800.0 PL=0
MOVL C02101 V=800.0 PL=0
MOVL C02102 V=800.0 PL=0
MOVL C02103 V=800.0 PL=0
MOVL C02104 V=800.0 PL=0
MOVL C02105 V=800.0 PL=0
MOVL C02106 V=800.0 PL=0
MOVL C02107 V=800.0 PL=0
MOVL C02108 V=800.0 PL=0
MOVL C02109 V=800.0 PL=0
MOVL C02110 V=800.0 PL=0
MOVL C02111 V=800.0 PL=0
MOVL C02112 V=800.0 PL=0
MOVL C02113 V=800.0 PL=0
MOVL C02114 V=800.0 PL=0
MOVL C02115 V=800.0 PL=0
MOVL C02116 V=800.0 PL=0
MOVL C02117 V=800.0 PL=0
MOVL C02118 V=800.0 PL=0
MOVL C02119 V=800.0 PL=0
MOVL C02120 V=800.0 PL=0
MOVL C02121 V=800.0 PL=0
MOVL C02122 V=800.0 PL=0
MOVL C02123 V=800.0 PL=0
MOVL C02124 V=800.0 PL=0
MOVL C02125 V=800.0 PL=0
MOVL C02126 V=800.0 PL=0
MOVL C02127 V=800.0 PL=0
MOVL C02128 V=800.0 PL=0
MOVL C02129 V=800.0 PL=0
MOVL C02130 V=800.0 PL=0
MOVL C02131 V=800.0 PL=0
MOVL C02132 V=800.0 PL=0
MOVL C02133 V=800.0 PL=0
MOVL C02134 V=800.0 PL=0
MOVL C02135 V=800.0 PL=0
MOVL C02136 V=800.0 PL=0
MOVL C02137 V=800.0 PL=0
MOVL C02138 V=800.0 PL=0
MOVL C02139 V=800.0 PL=0
MOVL C02140 V=800.0 PL=0
MOVL C02141 V=800.0 PL=0
MOVL C02142 V=800.0 PL=0
MOVL C02143 V=800.0 PL=0
MOVL C02144 V=800.0 PL=0
MOVL C02145 V=800.0 PL=0
MOVL C02146 V=800.0 PL=0
MOVL C02147 V=800.0 PL=0
MOVL C02148 V=800.0 PL=0
MOVL C02149 V=800.0 PL=0
MOVL C02150 V=800.0 PL=0
MOVL C02151 V=800.0 PL=0
MOVL C02152 V=800.0 PL=0
MOVL C02153 V=800.0 PL=0
MOVL C02154 V=800.0 PL=0
MOVL C02155 V=800.0 PL=0
MOVL C02156 V=800.0 PL=0
MOVL C02157 V=800.0 PL=0
MOVL C02158 V=800.0 PL=0
MOVL C02159 V=800.0 PL=0
MOVL C02160 V=800.0 PL=0
MOVL C02161 V=800.0 PL=0
MOVL C02162 V=800.0 PL=0
MOVL C02163 V=800.0 PL=0
MOVL C02164 V=800.0 PL=0
MOVL C02165 V=800.0 PL=0
